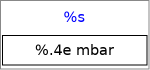
VISUALIZATION TEMPLATE_AMBIENT_PRESSURE_READING  // 150x70
VAR_IN_OUT
	m_instance: FB_METIS_AMBIENT_PRESSURE_SENSOR;
END_VAR
    Rectangle (2,35 145x30), "%.4e mbar", tooltip "Pressure in mbar", text variable: m_instance.stat.lrPressure, colour toggle: NOT m_instance.stat.bValid
    Rectangle (2,2 145x30), "%s", text variable: m_instance.in_sName
END_VISUALIZATION

// HMI/VISUs/Templates/TEMPLATE_BACKGROUND_LEVEL_2
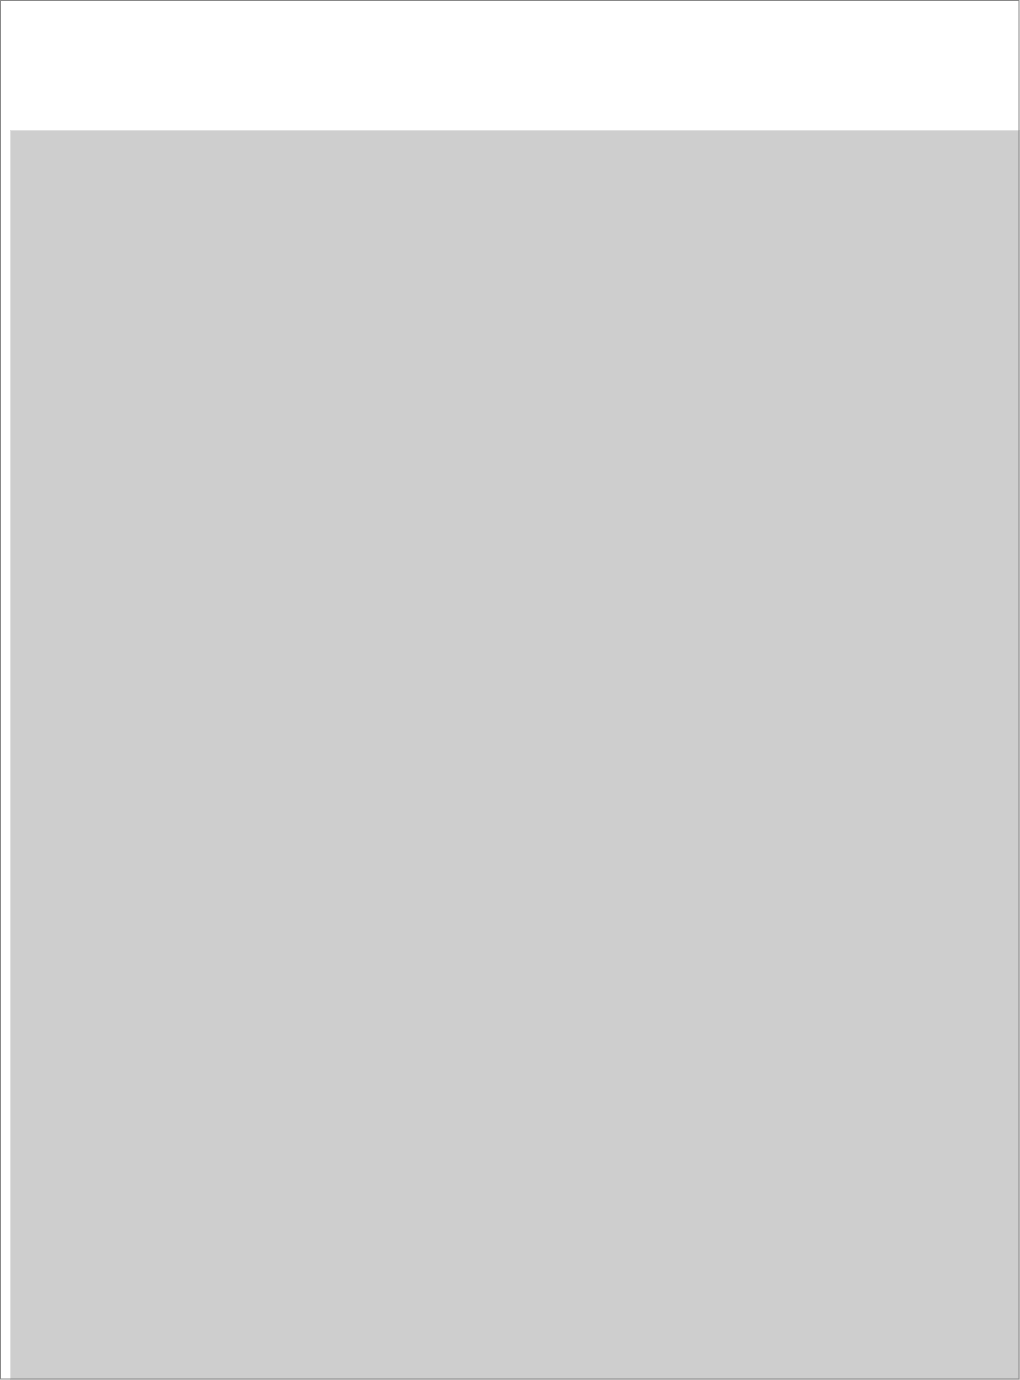
VISUALIZATION TEMPLATE_BACKGROUND_LEVEL_2  // 1020x1380
    Rectangle (10,130 1010x1250)
END_VISUALIZATION

// HMI/VISUs/Templates/TEMPLATE_BACKGROUND_LEVEL_3
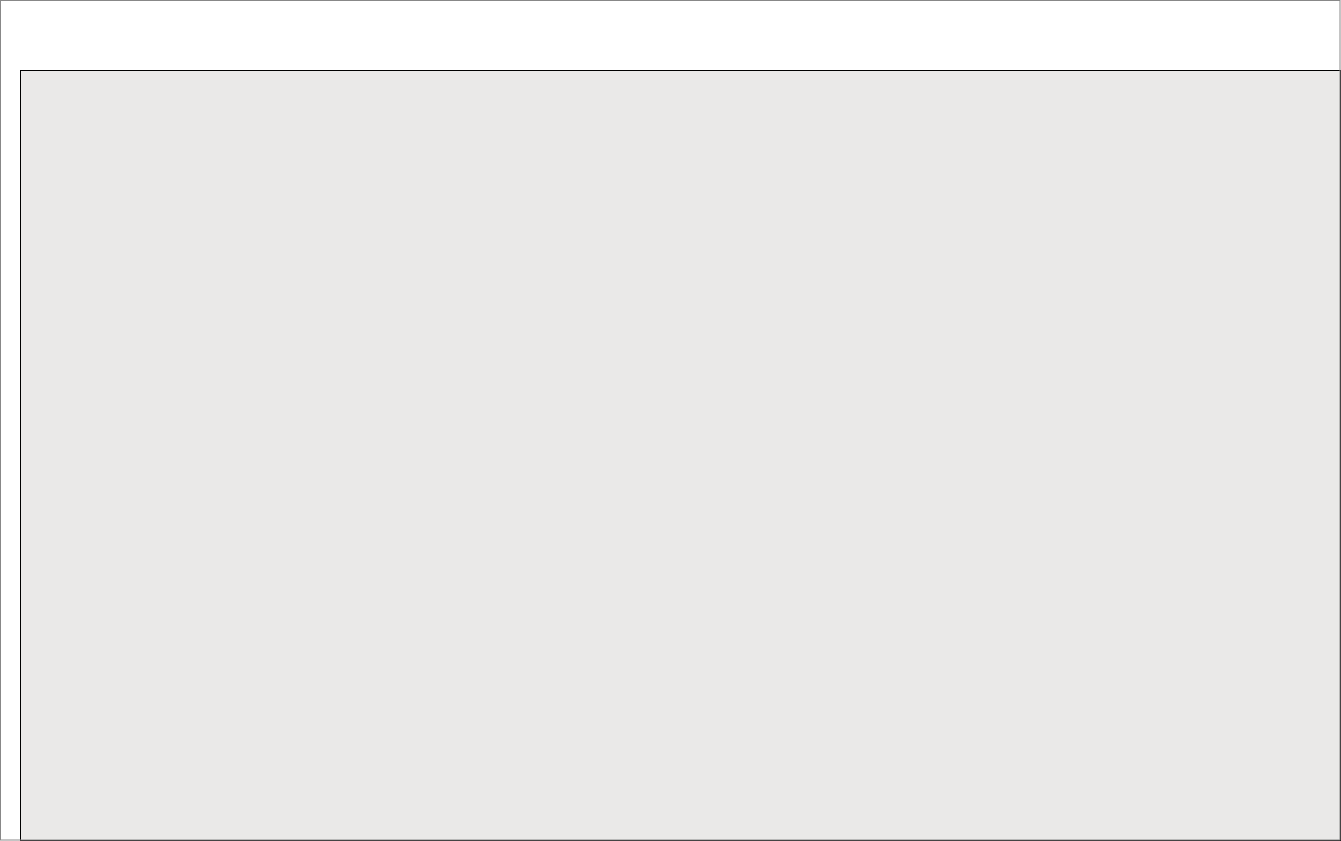
VISUALIZATION TEMPLATE_BACKGROUND_LEVEL_3  // 1341x841
    Rectangle (20,70 1321x771)
END_VISUALIZATION

// HMI/VISUs/Templates/TEMPLATE_BINARY_VALVES
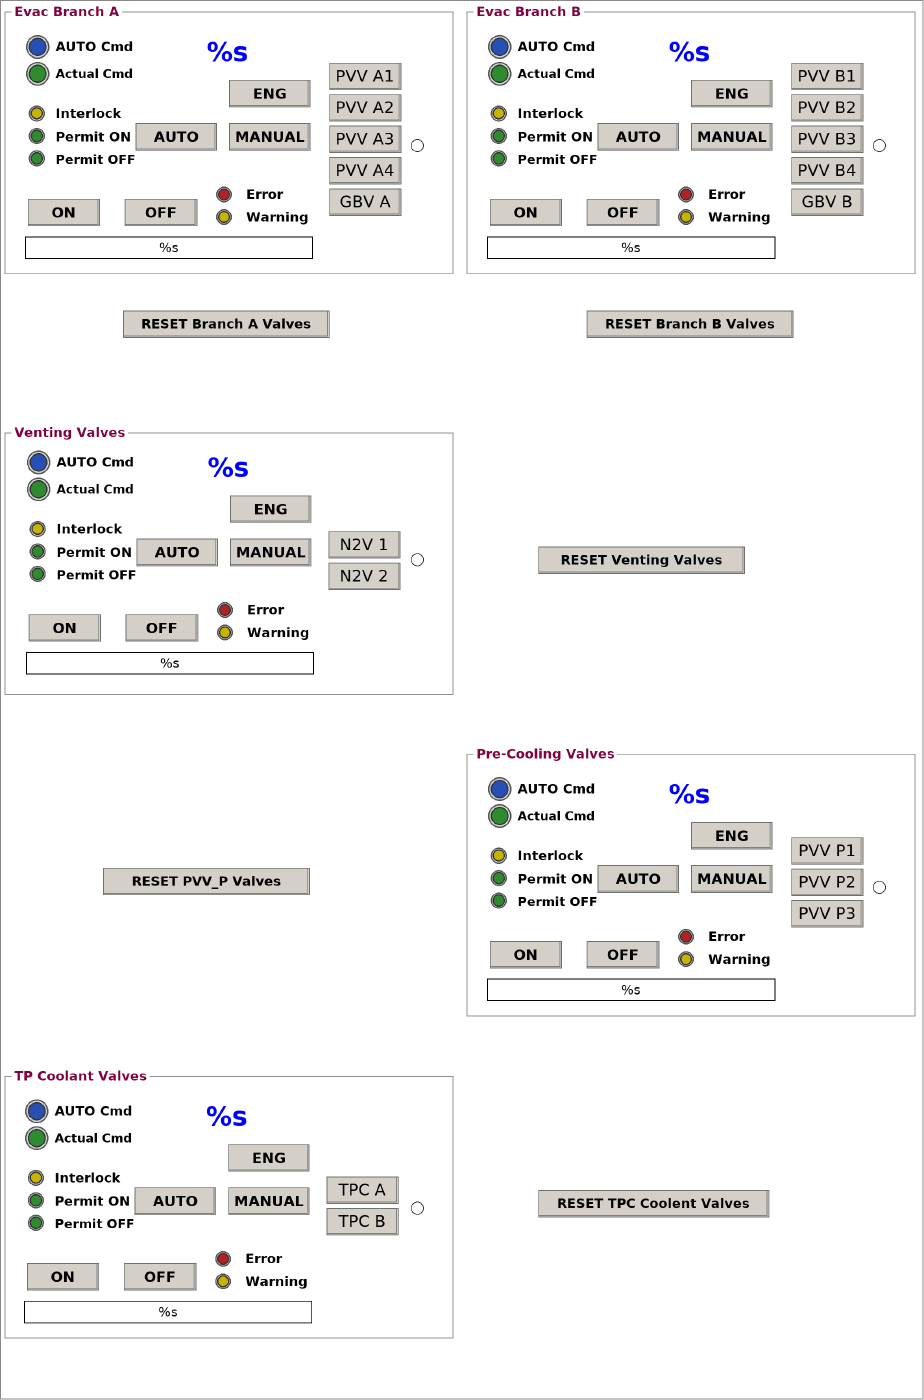
VISUALIZATION TEMPLATE_BINARY_VALVES  // 1030x1560
VAR_IN_OUT
	m_evac_Instance: FB_METIS_CRYO_EVAC;
	m_venting_instance:	FB_METIS_CRYO_VENTING;
	m_cool_down_instance: FB_METIS_CRYO_COOL_DOWN;
	m_cryo_instance:	FB_METIS_CRYO_CTRL;
	
END_VAR
    GroupBox (5,5 500x300), "Evac Branch A"
        Group (18,28 465x255)
            Group (344,37 121x181)
                Button (0,0 80x30), "PVV A1"
                    OnMouseClick: execute { m_evac_Instance.evac_branch_a.guiValveIndex := 1; }
                Button (0,35 80x30), "PVV A2"
                    OnMouseClick: execute { m_evac_Instance.evac_branch_a.guiValveIndex := 2; }
                Button (0,70 80x30), "PVV A3"
                    OnMouseClick: execute { m_evac_Instance.evac_branch_a.guiValveIndex := 3; }
                Button (0,105 80x30), "PVV A4"
                    OnMouseClick: execute { m_evac_Instance.evac_branch_a.guiValveIndex := 4; }
                Button (0,140 80x30), "GBV A"
                    OnMouseClick: execute { m_evac_Instance.evac_branch_a.guiValveIndex := 5; }
                RadioButton (89,3 32x178), variable: m_evac_Instance.evac_branch_a.guiValveIndex-1
            Frame (0,0 326x255)
                shows TEMPLATE_METIS_CMD_OVERRIDE(m_Cmd := m_evac_Instance.evac_branch_a.ptrVC[m_evac_Instance.evac_branch_a.guiValveIndex]^)
    GroupBox (520,5 500x300), "Evac Branch B"
        Group (18,28 465x255)
            Frame (0,0 326x255)
                shows TEMPLATE_METIS_CMD_OVERRIDE(m_Cmd := m_evac_Instance.evac_branch_b.ptrVC[m_evac_Instance.evac_branch_b.guiValveIndex]^)
            Group (344,37 121x181)
                Button (0,0 80x30), "PVV B1"
                    OnMouseClick: execute { m_evac_Instance.evac_branch_b.guiValveIndex := 1; }
                Button (0,35 80x30), "PVV B2"
                    OnMouseClick: execute { m_evac_Instance.evac_branch_b.guiValveIndex := 2; }
                Button (0,70 80x30), "PVV B3"
                    OnMouseClick: execute { m_evac_Instance.evac_branch_b.guiValveIndex := 3; }
                Button (0,105 80x30), "PVV B4"
                    OnMouseClick: execute { m_evac_Instance.evac_branch_b.guiValveIndex := 4; }
                Button (0,140 80x30), "GBV B"
                    OnMouseClick: execute { m_evac_Instance.evac_branch_b.guiValveIndex := 5; }
                RadioButton (89,3 32x178), variable: m_evac_Instance.evac_branch_b.guiValveIndex-1
    GroupBox (520,832 500x300), "Pre-Cooling Valves"
        Group (18,28 465x255)
            Frame (0,0 326x255)
                shows TEMPLATE_METIS_CMD_OVERRIDE(m_Cmd := m_cool_down_instance.ptrVC[m_cool_down_instance.guiValveIndex]^)
            Group (344,73 121x108)
                Button (0,0 80x30), "PVV P1"
                    OnMouseClick: execute { m_cool_down_instance.guiValveIndex := 1; }
                Button (0,35 80x30), "PVV P2"
                    OnMouseClick: execute { m_cool_down_instance.guiValveIndex := 2; }
                RadioButton (89,3 32x105), variable: m_cool_down_instance.guiValveIndex-1
                Button (0,70 80x30), "PVV P3"
                    OnMouseClick: execute { m_cool_down_instance.guiValveIndex := 3; }
    GroupBox (5,474 500x300), "Venting Valves"
        Group (19,22 462x255)
            Frame (0,0 326x255)
                shows TEMPLATE_METIS_CMD_OVERRIDE(m_Cmd := m_venting_instance.ptrVC[m_venting_instance.guiValveIndex]^)
            Group (342,94 120x67)
                Button (0,2 80x30), "N2V 1"
                    OnMouseClick: execute { m_venting_instance.guiValveIndex := 1; }
                Button (0,37 80x30), "N2V 2"
                    OnMouseClick: execute { m_venting_instance.guiValveIndex := 2; }
                RadioButton (90,0 30x67), variable: m_venting_instance.guiValveIndex-1
                    Areas[0]: Text=Radiobutton
                    Areas[1]: Text=Radiobutton
    GroupBox (5,1191 500x300), "TP Coolant Valves"
        Frame (17,28 326x255)
            shows TEMPLATE_METIS_CMD_OVERRIDE(m_Cmd := m_cryo_instance.ptrVC[m_cryo_instance.guiCoolantValveIndex]^)
        Group (359,120 124x70)
            Button (0,0 80x30), "TPC A"
                OnMouseClick: execute { m_cryo_instance.guiCoolantValveIndex := 1; }
            Button (0,35 80x30), "TPC B"
                OnMouseClick: execute { m_cryo_instance.guiCoolantValveIndex := 2; }
            RadioButton (92,0 32x70), variable: m_cryo_instance.guiCoolantValveIndex-1
    Button (137,346 230x30), "RESET Branch A Valves"
        OnMouseClick: execute { m_evac_Instance.evac_branch_a.bReset_Valves := TRUE; }
    Button (654,346 230x30), "RESET Branch B Valves"
        OnMouseClick: execute { m_evac_Instance.evac_branch_b.bReset_Valves := TRUE; }
    Button (600,609 230x30), "RESET Venting Valves"
        OnMouseClick: execute { m_venting_instance.bReset_Valves := TRUE; }
    Button (115,967 230x30), "RESET PVV_P Valves"
        OnMouseClick: execute { m_cool_down_instance.bReset_Valves := TRUE; }
    Button (600,1326 257x30), "RESET TPC Coolent Valves"
        OnMouseClick: execute { m_cryo_instance.TPC_A.M_Reset(); m_cryo_instance.TPC_B.M_Reset(); }
END_VISUALIZATION

// HMI/VISUs/Templates/TEMPLATE_CRYO_SENSOR_TEMPERATURE
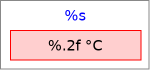
VISUALIZATION TEMPLATE_CRYO_SENSOR_TEMPERATURE  // 150x70
VAR_IN_OUT
	m_instance:	FB_CRYO_SENSOR_TEMPERATURE;
END_VAR
    Rectangle (10,30 131x30)
    Rectangle (10,30 131x30), invisible if: NOT m_instance.stat.bError
    Rectangle (10,30 131x31), "%.2f °C", text variable: m_instance.stat.lrTempC
    Rectangle (0,0 151x31), "%s", text variable: m_instance.in_sName
END_VISUALIZATION

// HMI/VISUs/Templates/TEMPLATE_EVACUATION
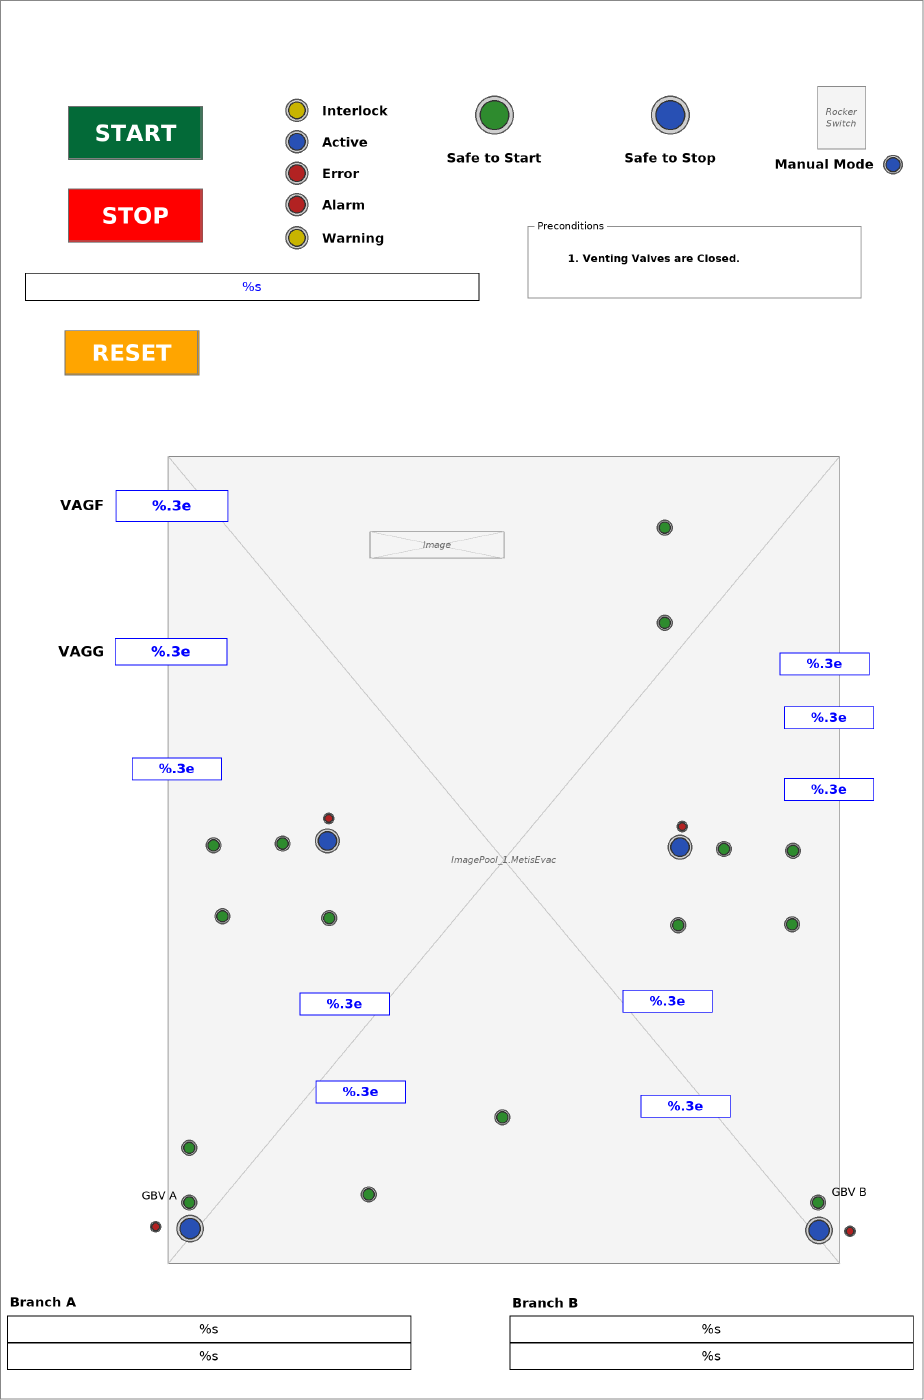
VISUALIZATION TEMPLATE_EVACUATION  // 1030x1560
VAR_IN_OUT
	m_Instance: FB_METIS_CRYO_EVAC;
	m_venting_instance:	FB_METIS_CRYO_VENTING;
	m_cool_down_instance: FB_METIS_CRYO_COOL_DOWN;
	
END_VAR
    Group (8,508 1010x1018)
        Group (0,928 1010x90)
            Group (0,0 450x90)
                Rectangle (0,30 450x30), "%s", text variable: m_Instance.evac_branch_a.stat.sErrorText
                Rectangle (0,60 450x30), "%s", text variable: m_Instance.evac_branch_a.stat.sStatus
                Rectangle (0,0 100x30), "Branch A"
            Group (560,1 450x89)
                Rectangle (0,29 450x30), "%s", text variable: m_Instance.evac_branch_b.stat.sErrorText
                Rectangle (0,59 450x30), "%s", text variable: m_Instance.evac_branch_b.stat.sStatus
                Rectangle (0,0 100x30), "Branch B"
        Group (45,0 921x900)
            Image (134,0 749x900), image: ImagePool_1.MetisEvac
            Image (359,84 150x30)
            Rectangle (281,598 100x25), "%.3e", text variable: m_Instance.evac_branch_a.VAG1.stat.lrPressure
            Rectangle (94,336 100x25), "%.3e", text variable: m_Instance.evac_branch_a.VAG2.stat.lrPressure
            Lamp1 (141,843 36x36), variable: m_Instance.evac_branch_a.rp.stat.bReady, style: Lamp-Lamp1-Blue
            Lamp1 (296,413 32x32), tooltip "If ON, TMP pump is at its nominal speed, i.e. Ready.", variable: m_Instance.evac_branch_a.tp.stat.bReady, style: Lamp-Lamp1-Blue
            Lamp1 (185,503 20x20), variable: m_Instance.evac_branch_a.PVV1.stat.bActON, style: Lamp-Lamp1-Green
            Lamp1 (304,505 20x20), variable: m_Instance.evac_branch_a.PVV2.stat.bActON, style: Lamp-Lamp1-Green
            Lamp1 (175,424 20x20), variable: m_Instance.evac_branch_a.PVV3.stat.bActON, style: Lamp-Lamp1-Green
            Lamp1 (252,422 20x20), variable: m_Instance.evac_branch_a.PVV4.stat.bActON, style: Lamp-Lamp1-Green
            Lamp1 (148,822 20x20), variable: m_Instance.evac_branch_a.GBV.stat.bActON, style: Lamp-Lamp1-Green
            Lamp1 (306,397 15x14), tooltip "If ON, TMP pump is still spinning.", variable: m_Instance.evac_branch_a.tp.stat.bSpeed100, style: Lamp-Lamp1-Red
            Rectangle (299,696 100x25), "%.3e", text variable: m_Instance.evac_branch_a.VAG3.stat.lrPressure
            Lamp1 (689,420 32x32), tooltip "If ON, TMP pump is at its nominal speed, i.e. Ready.", variable: m_Instance.evac_branch_b.tp.stat.bReady, style: Lamp-Lamp1-Blue
            Lamp1 (700,406 15x14), tooltip "If ON, TMP pump is still spinning.", variable: m_Instance.evac_branch_b.tp.stat.bSpeed100, style: Lamp-Lamp1-Red
            Lamp1 (744,428 20x20), variable: m_Instance.evac_branch_b.PVV4.stat.bActON, style: Lamp-Lamp1-Green
            Lamp1 (821,430 20x20), variable: m_Instance.evac_branch_b.PVV3.stat.bActON, style: Lamp-Lamp1-Green
            Lamp1 (693,513 20x20), variable: m_Instance.evac_branch_b.PVV2.stat.bActON, style: Lamp-Lamp1-Green
            Lamp1 (820,512 20x20), variable: m_Instance.evac_branch_b.PVV1.stat.bActON, style: Lamp-Lamp1-Green
            Lamp1 (842,845 36x36), variable: m_Instance.evac_branch_b.rp.stat.bReady, style: Lamp-Lamp1-Blue
            Lamp1 (849,822 20x20), variable: m_Instance.evac_branch_b.GBV.stat.bActON, style: Lamp-Lamp1-Green
            Rectangle (661,712 100x25), "%.3e", text variable: m_Instance.evac_branch_b.VAG3.stat.lrPressure
            Rectangle (821,359 100x25), "%.3e", text variable: m_Instance.evac_branch_b.VAG2.stat.lrPressure
            Rectangle (641,595 100x25), "%.3e", text variable: m_Instance.evac_branch_b.VAG1.stat.lrPressure
            Lamp1 (678,70 20x20), variable: m_venting_instance.N2V_1.stat.bActON, style: Lamp-Lamp1-Green
            Lamp1 (678,176 20x20), variable: m_venting_instance.N2V_2.stat.bActON, style: Lamp-Lamp1-Green
            Lamp1 (148,761 20x20), variable: m_cool_down_instance.PVV_P1.stat.bActON, style: Lamp-Lamp1-Green
            Lamp1 (348,813 20x20), variable: m_cool_down_instance.PVV_P3.stat.bActON, style: Lamp-Lamp1-Green
            Lamp1 (497,727 20x20), variable: m_cool_down_instance.PVV_P2.stat.bActON, style: Lamp-Lamp1-Green
            Rectangle (97,809 55x30), "GBV A"
            Rectangle (866,805 55x30), "GBV B"
            Group (1,38 200x35)
                Rectangle (75,0 125x35), "%.3e", text variable: m_Instance.VAGF.stat.lrPressure
                Rectangle (0,2 75x30), "VAGF"
            Group (0,203 200x30)
                Rectangle (75,0 125x30), "%.3e", text variable: m_Instance.VAGG.stat.lrPressure
                Rectangle (0,0 75x30), "VAGG"
            Rectangle (816,219 100x25), "%.3e", text variable: m_venting_instance.sensor_HPG1.stat.lrPressure
            Rectangle (821,279 100x25), "%.3e", text variable: m_venting_instance.sensor_HPG2.stat.lrPressure
    Group (76,118 150x152)
        Button (0,0 150x60), "START", input disabled if: NOT m_Instance.in_Cryo_Stat.bVentingValvesAreClosed
            OnMouseClick: execute { m_Instance.ctrl.bEnable := TRUE; }
        Button (0,92 150x60), "STOP", input disabled if: (NOT m_instance.in_Cryo_Stat.bPermitEvacuationStop) AND (NOT m_Instance.stat.bManual)
            OnMouseClick: execute { m_Instance.ctrl.bEnable := FALSE; }
    Group (316,108 131x173)
        Group (0,35 131x31)
            Label (40,0 91x31), "Active"
            Lamp1 (0,0 30x30), variable: m_Instance.stat.bActive, style: Lamp-Lamp1-Blue
        Group (0,70 130x31)
            Label (40,0 90x31), "Error"
            Lamp1 (0,0 30x30), variable: m_Instance.stat.bError, style: Lamp-Lamp1-Red
        Group (0,0 131x31)
            Lamp1 (0,0 30x30), variable: m_Instance.interlocks.bInterlock_Evacuation, style: Lamp-Lamp1-Yellow
            Label (40,0 91x31), "Interlock"
        Group (0,105 130x31)
            Label (40,0 90x31), "Alarm"
            Lamp1 (0,0 30x30), variable: m_Instance.stat.bAlarm, style: Lamp-Lamp1-Red
        Group (0,142 130x31)
            Label (40,0 90x31), "Warning"
            Lamp1 (0,0 30x30), variable: m_Instance.stat.bWarning, style: Lamp-Lamp1-Yellow
    Group (672,103 150x88)
        Lamp1 (50,0 50x50), variable: m_Instance.in_Cryo_Stat.bPermitEvacuationStop, style: Lamp-Lamp1-Blue
        Rectangle (0,58 150x30), "Safe to Stop"
    GroupBox (588,244 372x88), "Preconditions"
        Rectangle (42,29 300x30), "1. Venting Valves are Closed.", colour toggle: m_Instance.in_Cryo_Stat.bVentingValvesAreClosed
    Button (72,368 150x50), "RESET", invisible if: NOT m_Instance.stat.bError
        OnMouseClick: execute { m_Instance.ctrl.bReset := TRUE; }
    Rectangle (28,304 506x31), "%s", text variable: m_instance.stat.sState
    Group (868,168 140x30)
        Label (0,0 109x30), "Manual Mode"
        Lamp1 (115,3 25x25), variable: m_Instance.stat.bManual, style: Lamp-Lamp1-Blue
    RockerSwitch (911,96 54x70), tooltip "Activates the Manual mode", variable: m_Instance.stat.bManual, input disabled if: m_Instance.stat.bVentingValvesOpen, behaviour: TOGGLE, style: Switch-RockerSwitch-Red
    Group (476,103 150x88)
        Lamp1 (50,0 50x50), variable: NOT m_Instance.interlocks.bInterlock_Evacuation, style: Lamp-Lamp1-Green
        Rectangle (0,58 150x30), "Safe to Start"
    Lamp1 (940,1365 15x14), tooltip "If ON, RP pump is still spinning.", variable: m_Instance.evac_branch_b.rp.stat.bMoving, style: Lamp-Lamp1-Red
    Lamp1 (166,1360 15x14), tooltip "If ON, RP pump is still spinning.", variable: m_Instance.evac_branch_a.rp.stat.bMoving, style: Lamp-Lamp1-Red
END_VISUALIZATION

// HMI/VISUs/Templates/TEMPLATE_HEATER_CPAU60
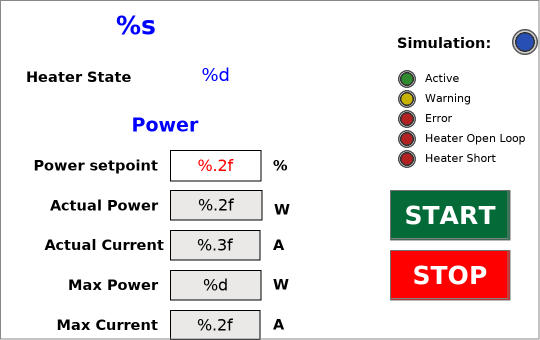
VISUALIZATION TEMPLATE_HEATER_CPAU60  // 540x340
VAR_IN_OUT
	m_instance: FB_HEATER_CPAU60;
	m_bEnable:	BOOL;	// Flag to start/stop the Heater
END_VAR
    Rectangle (21,10 230x30), "%s", text variable: m_Instance.in_sName
    Button (390,190 120x50), "START"
        OnMouseClick: execute { m_bEnable := TRUE; }
    Button (390,250 120x50), "STOP"
        OnMouseClick: execute { m_bEnable := FALSE; }
    Lamp1 (397,69 20x20), tooltip "If ON, Heater is active", variable: m_Instance.stat.bActive, style: Lamp-Lamp1-Green
    Lamp1 (397,89 20x20), tooltip "If ON, reading is in Warning", variable: m_Instance.stat.bWarning, style: Lamp-Lamp1-Yellow
    Lamp1 (397,129 20x20), tooltip "If ON, Heater circuit is open", variable: m_Instance.stat.bHeaterOpenLoop, style: Lamp-Lamp1-Red
    Lamp1 (397,149 20x20), tooltip "If ON, Heater is in short circuit", variable: m_Instance.stat.bHeaterShort, style: Lamp-Lamp1-Red
    Lamp1 (397,109 20x20), tooltip "If ON, reading is in error.", variable: m_Instance.stat.bError, style: Lamp-Lamp1-Red
    Label (422,67 87x23), "Active"
    Label (422,87 87x23), "Warning"
    Label (422,107 87x23), "Error"
    Label (422,127 112x23), "Heater Open Loop"
    Label (422,147 87x23), "Heater Short"
    Rectangle (170,150 91x31), "%.2f", tooltip "Simulated value [K] when simulation is active.", text variable: m_instance.ctrl.lrPower, input disabled if: Not m_instance.bManualInputFlag
        OnMouseClick: write the text variable via Default
    Rectangle (170,190 92x30), "%.2f", tooltip "Value used by the system [K]", text variable: m_instance.stat.lrActHeaterPower
    Rectangle (170,230 90x30), "%.3f", tooltip "Value used by the system [C]", text variable: m_instance.stat.lrActCurrent
    Lamp1 (510,27 30x30), tooltip "If ON, Heater is simulated.", variable: m_instance.stat.bSimulated, style: Lamp-Lamp1-Blue
    Rectangle (394,28 110x30), "Simulation:"
    Rectangle (90,110 150x30), "Power"
    Rectangle (271,195 29x29), "W"
    Rectangle (270,230 32x30), "A"
    Rectangle (138,60 156x30), "%d", text variable: m_Instance.stat.nHeaterState
    Rectangle (23,62 110x30), "Heater State"
    Rectangle (30,150 131x31), "Power setpoint"
    Rectangle (50,190 111x31), "Actual Power"
    Rectangle (270,150 29x31), "%"
    Rectangle (40,230 127x30), "Actual Current"
    Rectangle (170,270 91x30), "%d", tooltip "Value used by the system [K]", text variable: m_instance.in_nMaxHeaterPower
    Rectangle (170,310 90x30), "%.2f", tooltip "Value used by the system [K]", text variable: m_instance.stat.lrMaxCurrent
    Rectangle (60,270 101x30), "Max Power"
    Rectangle (30,310 131x30), "Max Current"
    Rectangle (270,270 29x29), "W"
    Rectangle (270,310 29x29), "A"
END_VISUALIZATION

// HMI/VISUs/Templates/TEMPLATE_HEATER_CXWUI60
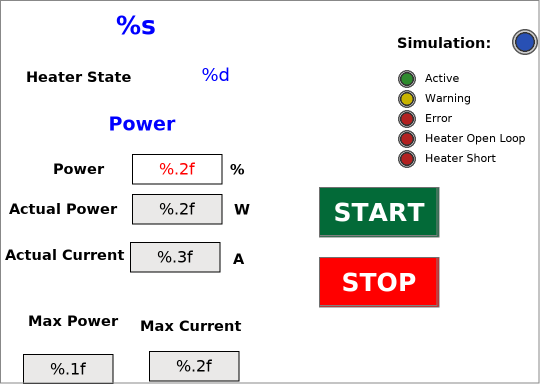
VISUALIZATION TEMPLATE_HEATER_CXWUI60  // 540x384
VAR_IN_OUT
	m_instance: FB_HEATER_CXWUI60;
	m_bEnable:	BOOL;	// Flag to start/stop the Heater
END_VAR
    Rectangle (21,10 230x30), "%s", text variable: m_Instance.in_sName
    Button (319,187 120x50), "START"
        OnMouseClick: execute { m_bEnable := TRUE; }
    Button (319,257 120x50), "STOP"
        OnMouseClick: execute { m_bEnable := FALSE; }
    Lamp1 (397,69 20x20), tooltip "If ON, Heater is active", variable: m_Instance.stat.bActive, style: Lamp-Lamp1-Green
    Lamp1 (397,89 20x20), tooltip "If ON, reading is in Warning", variable: m_Instance.stat.bWarning, style: Lamp-Lamp1-Yellow
    Lamp1 (397,129 20x20), tooltip "If ON, Heater circuit is open", variable: m_Instance.stat.bHeaterOpenLoop, style: Lamp-Lamp1-Red
    Lamp1 (397,149 20x20), tooltip "If ON, Heater is in short circuit", variable: m_Instance.stat.bHeaterShort, style: Lamp-Lamp1-Red
    Lamp1 (397,109 20x20), tooltip "If ON, reading is in error.", variable: m_Instance.stat.bError, style: Lamp-Lamp1-Red
    Label (422,67 87x23), "Active"
    Label (422,87 87x23), "Warning"
    Label (422,107 87x23), "Error"
    Label (422,127 112x23), "Heater Open Loop"
    Label (422,147 87x23), "Heater Short"
    Rectangle (132,154 90x30), "%.2f", tooltip "Simulated value [K] when simulation is active.", text variable: m_instance.ctrl.lrPower, input disabled if: Not m_instance.bManualInputFlag
        OnMouseClick: write the text variable via Default
    Rectangle (132,194 90x30), "%.2f", tooltip "Value used by the system [K]", text variable: m_instance.stat.lrActHeaterPower
    Rectangle (130,242 90x30), "%.3f", tooltip "Value used by the system [C]", text variable: m_instance.stat.lrActCurrent
    Lamp1 (510,27 30x30), tooltip "If ON, Heater is simulated.", style: Lamp-Lamp1-Blue
    Rectangle (394,28 110x30), "Simulation:"
    Rectangle (67,109 150x30), "Power"
    Rectangle (231,195 29x29), "W"
    Rectangle (230,244 32x30), "A"
    Rectangle (138,60 156x30), "%d", text variable: m_Instance.stat.nHeaterState
    Rectangle (23,62 110x30), "Heater State"
    Rectangle (50,154 66x30), "Power"
    Rectangle (6,194 110x30), "Actual Power"
    Rectangle (227,155 29x29), "%"
    Rectangle (2,240 127x30), "Actual Current"
    Rectangle (23,354 90x30), "%.1f", tooltip "Value used by the system [K]", text variable: m_instance.in_nMaxHeaterPower
    Rectangle (149,351 90x30), "%.2f", tooltip "Value used by the system [K]", text variable: m_instance.stat.lrMaxCurrent
    Rectangle (25,306 92x30), "Max Power"
    Rectangle (137,311 127x30), "Max Current"
END_VISUALIZATION

// HMI/VISUs/Templates/TEMPLATE_HEATER_PWM_CTRL
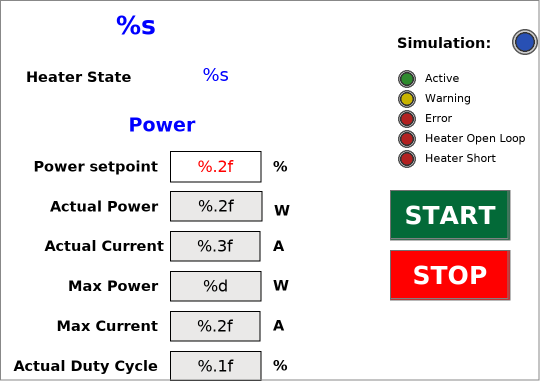
VISUALIZATION TEMPLATE_HEATER_PWM_CTRL  // 540x381
VAR_IN_OUT
	m_instance: FB_HEATER_PWM;
	m_bEnable:	BOOL;	// Flag to start/stop the Heater
END_VAR
    Rectangle (170,351 91x30), "%.1f", tooltip "Value used by the system [C]", text variable: m_instance.stat.lrActDutyCycle
    Rectangle (10,351 151x30), "Actual Duty Cycle"
    Rectangle (21,10 230x30), "%s", text variable: m_Instance.in_sName
    Button (390,190 120x50), "START"
        OnMouseClick: execute { m_bEnable := TRUE; }
    Button (390,250 120x50), "STOP"
        OnMouseClick: execute { m_bEnable := FALSE; }
    Lamp1 (397,69 20x20), tooltip "If ON, Heater is active", variable: m_Instance.stat.bActive, style: Lamp-Lamp1-Green
    Lamp1 (397,89 20x20), tooltip "If ON, reading is in Warning", variable: m_Instance.stat.bWarning, style: Lamp-Lamp1-Yellow
    Lamp1 (397,129 20x20), tooltip "If ON, Heater circuit is open", variable: m_Instance.stat.bHeaterOpenLoop, style: Lamp-Lamp1-Red
    Lamp1 (397,149 20x20), tooltip "If ON, Heater is in short circuit", variable: m_Instance.stat.bHeaterShort, style: Lamp-Lamp1-Red
    Lamp1 (397,109 20x20), tooltip "If ON, reading is in error.", variable: m_Instance.stat.bError, style: Lamp-Lamp1-Red
    Label (422,67 87x23), "Active"
    Label (422,87 87x23), "Warning"
    Label (422,107 87x23), "Error"
    Label (422,127 112x23), "Heater Open Loop"
    Label (422,147 87x23), "Heater Short"
    Rectangle (170,151 91x31), "%.2f", tooltip "Simulated value [K] when simulation is active.", text variable: m_instance.ctrl.lrPower, input disabled if: Not m_instance.bManualInputFlag
        OnMouseClick: write the text variable via Default
    Rectangle (170,191 92x30), "%.2f", tooltip "Value used by the system [K]", text variable: m_instance.stat.lrActHeaterPower
    Rectangle (170,231 90x30), "%.3f", tooltip "Value used by the system [C]", text variable: m_instance.stat.lrActCurrent
    Lamp1 (510,27 30x30), tooltip "If ON, Heater is simulated.", variable: m_instance.stat.bSimulated, style: Lamp-Lamp1-Blue
    Rectangle (394,28 110x30), "Simulation:"
    Rectangle (87,110 150x30), "Power"
    Rectangle (271,196 29x29), "W"
    Rectangle (270,231 32x30), "A"
    Rectangle (138,60 156x30), "%s", text variable: m_Instance.stat.sHeaterState
    Rectangle (23,62 110x30), "Heater State"
    Rectangle (30,151 131x31), "Power setpoint"
    Rectangle (50,191 111x31), "Actual Power"
    Rectangle (270,151 29x31), "%"
    Rectangle (40,231 127x30), "Actual Current"
    Rectangle (170,271 91x30), "%d", tooltip "Value used by the system [K]", text variable: m_instance.in_nMaxHeaterPower
    Rectangle (170,311 90x30), "%.2f", tooltip "Value used by the system [K]", text variable: m_instance.stat.lrMaxCurrent
    Rectangle (60,271 101x30), "Max Power"
    Rectangle (30,311 131x30), "Max Current"
    Rectangle (270,271 29x29), "W"
    Rectangle (270,311 29x29), "A"
    Rectangle (270,350 29x31), "%"
END_VISUALIZATION

// HMI/VISUs/Templates/TEMPLATE_LN2_LEVEL_SENSOR_AND_CTRL
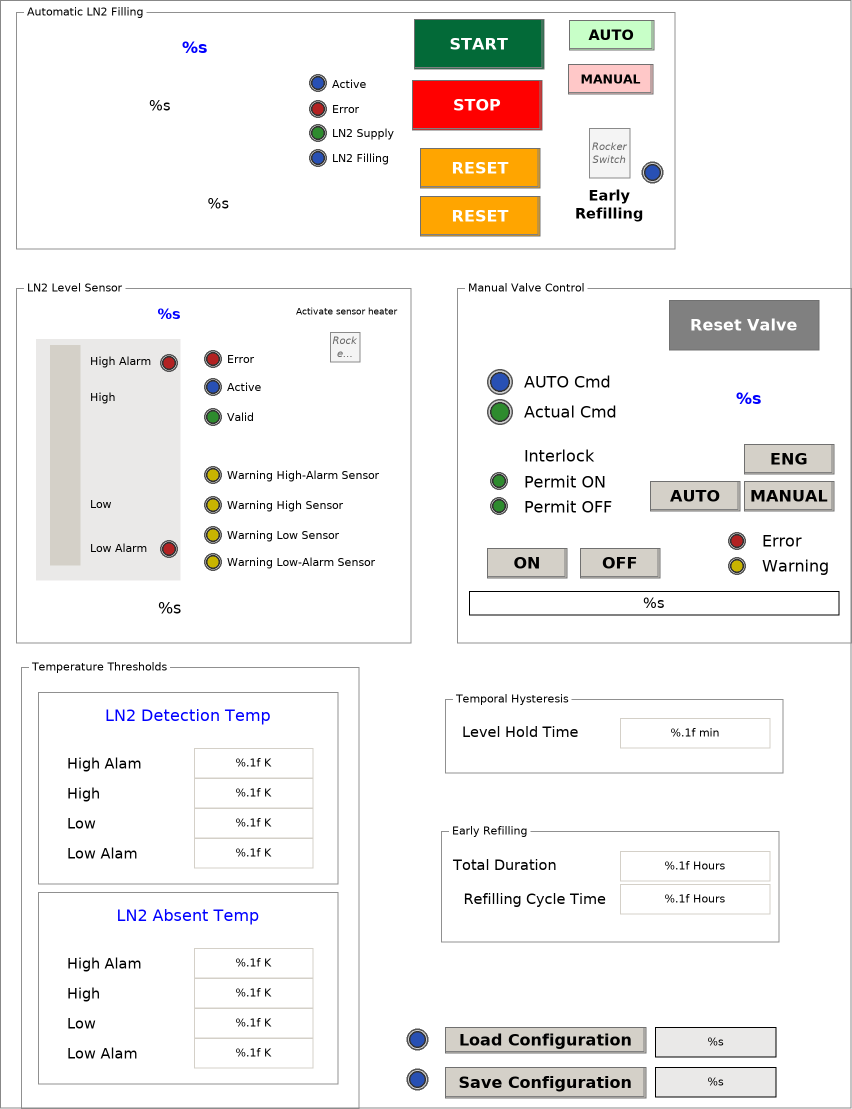
VISUALIZATION TEMPLATE_LN2_LEVEL_SENSOR_AND_CTRL  // 852x1109
VAR_IN_OUT
	m_level_control_instance: FB_METIS_CRYO_LN2_LEVEL_CTRL;
	m_instance: FB_METIS_CRYO_LN2_SENSOR;
	m_cmd: FB_CRYO_CMD_OVERRIDE;
	m_bEnable:	BOOL;	// Flag to start/stop LN2 level control
END_VAR
    GroupBox (457,280 395x363), "Manual Valve Control"
        Button (212,20 150x50), "Reset Valve", tooltip "Reset LN2 filling valve"
            OnMouseClick: execute { m_level_control_instance.M_ResetValve(); }
    Group (469,367 370x248)
        Lamp1 (20,104 20x20), variable: m_Cmd.bPermitOn, style: Lamp-Lamp1-Green
        Lamp1 (20,129 20x20), variable: m_Cmd.bPermitOff, style: Lamp-Lamp1-Green
        Rectangle (52,74 110x30), "Interlock"
        Rectangle (52,100 110x30), "Permit ON"
        Rectangle (52,125 110x30), "Permit OFF"
        Button (18,181 80x30), "ON", colour toggle: (m_Cmd.bPermitOn AND NOT m_Cmd.bAutoMode) OR m_Cmd.bEngMode, input disabled if: m_Cmd.bDisableBtnOn
            OnMouseClick: execute { m_Cmd.bManualCmd := TRUE; }
        Lamp1 (16,30 30x30), tooltip "Actual command going out", variable: m_Cmd.out_bEnable, style: Lamp-Lamp1-Green
        Rectangle (52,30 110x30), "Actual Cmd"
        Button (181,114 90x30), "AUTO", tooltip "Switch to AUTO Mode", colour toggle: m_Cmd.bAutoMode, input disabled if: m_Cmd.bAutoMode OR m_Cmd.bEngMode
            OnMouseClick: execute { m_Cmd.bAutoMode := TRUE; }
        Button (275,114 90x30), "MANUAL", tooltip "Switch to MANUAL Mode", colour toggle: NOT m_Cmd.bAutoMode, input disabled if: NOT m_Cmd.bAutoMode AND NOT m_Cmd.bEngMode
            OnMouseClick: execute { m_Cmd.bAutoMode := FALSE; }
        Button (111,181 80x30), "OFF", colour toggle: (m_Cmd.bPermitOff AND NOT m_Cmd.bAutoMode) OR m_Cmd.bEngMode, input disabled if: m_Cmd.bDisableBtnOff
            OnMouseClick: execute { m_Cmd.bManualCmd := FALSE; }
        Button (275,77 90x30), "ENG", tooltip "Toggle Engineering Mode", colour toggle: m_Cmd.bEngMode, input disabled if: m_Cmd.bAutoMode
            toggle m_Cmd.bEngMode
        Lamp1 (16,0 30x30), tooltip "Command coming from the Control System", variable: m_Cmd.in_bEnable, style: Lamp-Lamp1-Blue
        Rectangle (52,0 110x30), "AUTO Cmd"
        Rectangle (0,224 370x24), "%s", text variable: m_Cmd.out_sStatus
        Lamp1 (258,164 20x20), tooltip "If ON, there is an error in the SW implementation of permission handling.", variable: m_Cmd.out_bError, style: Lamp-Lamp1-Red
        Rectangle (290,159 75x30), "Error"
        Lamp1 (258,189 20x20), tooltip "If ON, ENG command is not safe!", variable: m_Cmd.out_bWarning, style: Lamp-Lamp1-Yellow
        Rectangle (290,184 75x30), "Warning"
        Rectangle (205,11 150x41), "%s", text variable: m_Cmd.out_sMode
    GroupBox (441,823 338x119), "Early Refilling", tooltip "Time to hold a change of status to avoid transient oscillations."
        Label (9,59 170x34), "Refilling Cycle Time"
        Textfield (179,61 150x30), "%.1f Hours", tooltip "(Hours) Refilling cycle time during the Early refilling", text variable: m_level_control_instance.cfg.lr_Cycle_Time, input disabled if: m_level_control_instance.bAuto
            OnMouseClick: write the text variable via Default
        Textfield (179,28 150x30), "%.1f Hours", tooltip "(Hours) The total duration of Early Refilling", text variable: m_level_control_instance.cfg.lr_Early_Refill_Duration_Time, input disabled if: m_level_control_instance.bAuto
            OnMouseClick: write the text variable via Default
        Label (9,25 170x34), "Total Duration"
    GroupBox (445,691 338x82), "Temporal Hysteresis", tooltip "Time to hold a change of status to avoid transient oscillations."
        Textfield (175,27 150x30), "%.1f min", tooltip "(Minutes) LN2 level hold time to reduce oscilations at level change", text variable: m_level_control_instance.cfg.lr_LN2Level_Hold_Time, input disabled if: m_level_control_instance.bAuto
            OnMouseClick: write the text variable via Default
        Label (14,24 158x34), "Level Hold Time"
    GroupBox (16,4 659x245), "Automatic LN2 Filling"
        Rectangle (12,74 264x55), "%s", text variable: m_level_control_instance.sState
        Label (313,69 46x23), "Active"
        Lamp1 (292,95 20x20), tooltip "pump speed > 0 rpm", variable: m_level_control_instance.bError, style: Lamp-Lamp1-Red
        Label (313,94 46x23), "Error"
        Lamp1 (292,69 20x20), tooltip "pump speed > 0 rpm", variable: m_level_control_instance.bActive, style: Lamp-Lamp1-Blue
        Lamp1 (292,119 20x20), tooltip "pump speed > 0 rpm", variable: m_level_control_instance.in_ESO_LN2_Supply, style: Lamp-Lamp1-Green
        Button (553,16 85x30), "AUTO", tooltip "Automatic LN2 Level Control", colour toggle: m_level_control_instance.bAuto
            OnMouseClick: execute { m_level_control_instance.bManual := FALSE; m_level_control_instance.bAuto := TRUE; }
        Button (552,60 85x30), "MANUAL", tooltip "Manually start/Stop LN2 Level Control", colour toggle: m_level_control_instance.bManual
            OnMouseClick: execute { m_level_control_instance.bManual := TRUE; m_level_control_instance.bAuto := FALSE; }
        Group (552,124 83x97)
            RockerSwitch (21,0 41x50), tooltip "Activate or deactivate early LN2 refilling", variable: m_level_control_instance.bEarly_Refilling, behaviour: TOGGLE, style: Switch-RockerSwitch-Blue
            Label (0,56 83x41), "Early Refilling"
        Button (404,144 120x40), "RESET"
            OnMouseClick: execute {
                m_level_control_instance.nState := E_LN2_LEVEL_CTRL_STATE.ERROR; // RESET
                m_level_control_instance.bReset := TRUE;
            }
        Button (404,192 120x40), "RESET", invisible if: NOT m_level_control_instance.bError
            OnMouseClick: execute { m_level_control_instance.bReset := TRUE; }
        Rectangle (12,172 381x55), "%s", text variable: m_level_control_instance.sSubState
        Lamp1 (292,144 20x20), tooltip "pump speed > 0 rpm", variable: m_level_control_instance.bFilling, style: Lamp-Lamp1-Blue
        Lamp1 (624,156 25x25), tooltip "pump speed > 0 rpm", variable: m_level_control_instance.bEarly_Refilling, style: Lamp-Lamp1-Blue
    GroupBox (16,280 395x363), "LN2 Level Sensor", tooltip "LN2 Level Sensor"
        RockerSwitch (314,52 30x30), tooltip "Activate or deactivate sensor heaters", variable: m_instance.bActivateSensor, behaviour: TOGGLE, style: Switch-RockerSwitch-Yellow
        Label (277,16 111x31), "Activate sensor heater"
    Rectangle (37,299 264x30), "%s", text variable: m_instance.in_sName
    Rectangle (36,339 144x241)
    Group (50,345 30x220)
        Rectangle (0,180 30x40), colour toggle: m_instance.stat.bLowAlarm
        Rectangle (0,110 30x70), colour toggle: m_instance.stat.bLow
        Rectangle (0,40 30x70), colour toggle: m_instance.stat.bHigh
        Rectangle (0,0 30x40), colour toggle: m_instance.stat.bHighAlarm
    Label (87,350 70x23), "High Alarm"
    Label (87,386 34x23), "High"
    Label (87,493 28x23), "Low"
    Label (87,537 70x23), "Low Alarm"
    Lamp1 (159,353 20x20), variable: m_instance.stat.bLowAlarm AND ( m_instance.stat.bLow) AND ( m_instance.stat.bHigh) AND (m_instance.stat.bHighAlarm), style: Lamp-Lamp1-Red
    Lamp1 (159,539 20x20), variable: m_instance.stat.bLowAlarm AND (NOT m_instance.stat.bLow) AND (NOT m_instance.stat.bHigh) AND (NOT m_instance.stat.bHighAlarm), style: Lamp-Lamp1-Red
    Lamp1 (203,407 20x20), tooltip "If ON, reading is valid.", variable: m_instance.stat.bValid, style: Lamp-Lamp1-Green
    Label (224,406 44x23), "Valid"
    Lamp1 (203,377 20x20), tooltip "pump speed > 0 rpm", variable: m_Instance.stat.bActive, style: Lamp-Lamp1-Blue
    Label (224,376 46x23), "Active"
    Lamp1 (203,495 20x20), tooltip "If ON, reading is valid.", variable: m_instance.stat.bWarningSens_H, style: Lamp-Lamp1-Yellow
    Label (224,494 156x23), "Warning High Sensor"
    Lamp1 (203,465 20x20), tooltip "pump speed > 0 rpm", variable: m_Instance.stat.bWarningSens_HA, style: Lamp-Lamp1-Yellow
    Label (224,464 166x23), "Warning High-Alarm Sensor"
    Lamp1 (203,525 20x20), tooltip "If ON, reading is valid.", variable: m_instance.stat.bWarningSens_L, style: Lamp-Lamp1-Yellow
    Label (224,524 125x23), "Warning Low Sensor"
    Lamp1 (203,552 20x20), tooltip "If ON, reading is valid.", variable: m_instance.stat.bWarningSens_LA, style: Lamp-Lamp1-Yellow
    Label (224,551 164x23), "Warning Low-Alarm Sensor"
    Rectangle (38,593 264x30), "%s", text variable: m_instance.stat.sStatus
    Lamp1 (203,349 20x20), tooltip "pump speed > 0 rpm", variable: m_Instance.stat.bError, style: Lamp-Lamp1-Red
    Label (224,348 46x23), "Error"
    Button (414,19 130x50), "START", input disabled if: m_level_control_instance.bAuto
        OnMouseClick: execute { m_bEnable := TRUE; }
    Button (412,80 130x50), "STOP", input disabled if: m_level_control_instance.bAuto
        OnMouseClick: execute { m_bEnable := FALSE; }
    Rectangle (28,26 334x43), "%s", tooltip "LN2 level control", text variable: m_level_control_instance.in_sName
    Label (329,122 67x23), "LN2 Supply"
    GroupBox (21,659 338x450), "Temperature Thresholds", tooltip "Temp thresholds for LN2 detection and temperature hysteresis"
    GroupBox (38,684 300x200)
    Label (89,701 198x29), "LN2 Detection Temp"
    Textfield (194,748 119x30), "%.1f K", tooltip "LN2 detection temperature threshold", text variable: m_level_control_instance.cfg.lrLN2_Level_SenseTempK_HA, input disabled if: m_level_control_instance.bAuto
        OnMouseClick: write the text variable via Default
    Label (64,749 100x29), "High Alam"
    Textfield (194,778 119x30), "%.1f K", tooltip "LN2 detection temperature threshold", text variable: m_level_control_instance.cfg.lrLN2_Level_SenseTempK_H, input disabled if: m_level_control_instance.bAuto
        OnMouseClick: write the text variable via Default
    Label (64,779 100x29), "High"
    Textfield (194,808 119x30), "%.1f K", tooltip "LN2 detection temperature threshold", text variable: m_level_control_instance.cfg.lrLN2_Level_SenseTempK_L, input disabled if: m_level_control_instance.bAuto
        OnMouseClick: write the text variable via Default
    Label (64,809 100x29), "Low"
    Textfield (194,838 119x30), "%.1f K", tooltip "LN2 detection temperature threshold", text variable: m_level_control_instance.cfg.lrLN2_Level_SenseTempK_LA, input disabled if: m_level_control_instance.bAuto
        OnMouseClick: write the text variable via Default
    Label (64,839 100x29), "Low Alam"
    GroupBox (38,884 300x200)
    Label (89,901 198x29), "LN2 Absent Temp"
    Textfield (194,948 119x30), "%.1f K", tooltip "LN2 detection temperature threshold", text variable: m_level_control_instance.cfg.lrLN2_Level_AbsenceTempK_HA, input disabled if: m_level_control_instance.bAuto
        OnMouseClick: write the text variable via Default
    Label (64,949 100x29), "High Alam"
    Textfield (194,978 119x30), "%.1f K", tooltip "LN2 detection temperature threshold", text variable: m_level_control_instance.cfg.lrLN2_Level_AbsenceTempK_H, input disabled if: m_level_control_instance.bAuto
        OnMouseClick: write the text variable via Default
    Label (64,979 100x29), "High"
    Textfield (194,1008 119x30), "%.1f K", tooltip "LN2 detection temperature threshold", text variable: m_level_control_instance.cfg.lrLN2_Level_AbsenceTempK_L, input disabled if: m_level_control_instance.bAuto
        OnMouseClick: write the text variable via Default
    Label (64,1009 100x29), "Low"
    Textfield (194,1038 119x30), "%.1f K", tooltip "LN2 detection temperature threshold", text variable: m_level_control_instance.cfg.lrLN2_Level_AbsenceTempK_LA, input disabled if: m_level_control_instance.bAuto
        OnMouseClick: write the text variable via Default
    Label (64,1039 100x29), "Low Alam"
    Lamp1 (405,1027 25x25), tooltip "Command coming from the Control System", variable: m_level_control_instance.ctrl.bReadConfig, style: Lamp-Lamp1-Blue
    Button (445,1067 201x31), "Save Configuration", input disabled if: m_level_control_instance.bAuto
        OnMouseClick: execute { m_level_control_instance.ctrl.bWriteConfig := TRUE; }
    Button (445,1027 201x26), "Load Configuration", input disabled if: m_level_control_instance.bAuto
        OnMouseClick: execute { m_level_control_instance.ctrl.bReadConfig := TRUE; }
    Lamp1 (405,1067 25x25), tooltip "Command coming from the Control System", variable: m_level_control_instance.ctrl.bWriteConfig, style: Lamp-Lamp1-Blue
    Rectangle (655,1027 121x30), "%s", text variable: m_level_control_instance.fbConfig.sReadError, colour toggle: m_level_control_instance.fbConfig.bReadError
    Rectangle (655,1067 121x30), "%s", text variable: m_level_control_instance.fbConfig.sWriteError, colour toggle: m_level_control_instance.fbConfig.bWriteError
    Label (329,147 72x23), "LN2 Filling"
END_VISUALIZATION

// HMI/VISUs/Templates/TEMPLATE_MAIN_FSM
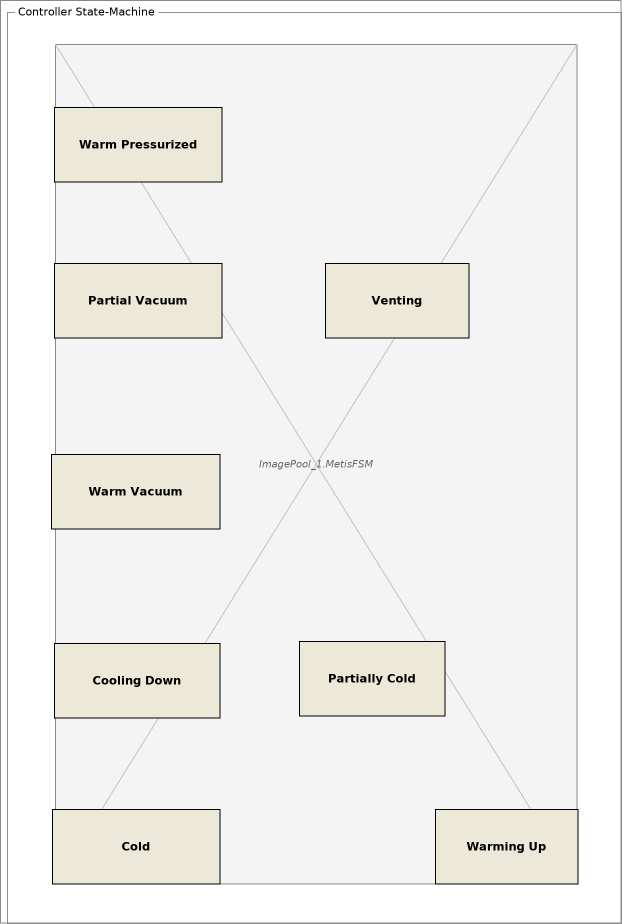
VISUALIZATION TEMPLATE_MAIN_FSM  // 622x924
VAR_IN_OUT
	m_instance:	FB_METIS_CRYO_CTRL;
END_VAR
    GroupBox (7,4 615x920), "Controller State-Machine"
    Group (51,44 527x840)
        Image (4,0 522x840), image: ImagePool_1.MetisFSM
        RoundedRectangle (1,765 168x75), "Cold", colour toggle: m_instance.stat.nState = E_METIS_CRYO_CTRL_STATE.COLD
        RoundedRectangle (3,599 166x75), "Cooling Down", colour toggle: m_instance.stat.nState = E_METIS_CRYO_CTRL_STATE.COOLING_DOWN
        RoundedRectangle (384,765 143x75), "Warming Up", colour toggle: m_instance.stat.nState = E_METIS_CRYO_CTRL_STATE.WARMING_UP
        RoundedRectangle (274,219 144x75), "Venting", colour toggle: m_instance.stat.nState = E_METIS_CRYO_CTRL_STATE.VENTING
        RoundedRectangle (0,410 169x75), "Warm Vacuum", colour toggle: m_instance.stat.nState = E_METIS_CRYO_CTRL_STATE.WARM_VACUUM
        RoundedRectangle (3,63 168x75), "Warm Pressurized", colour toggle: m_instance.stat.nState = E_METIS_CRYO_CTRL_STATE.WARM_PRESS
        RoundedRectangle (3,219 168x75), "Partial Vacuum", colour toggle: m_instance.stat.nState = E_METIS_CRYO_CTRL_STATE.PARTIAL_VACUUM
        RoundedRectangle (248,597 146x75), "Partially Cold", colour toggle: m_instance.stat.nState = E_METIS_CRYO_CTRL_STATE.PARTIALLY_COLD
END_VISUALIZATION

// HMI/VISUs/Templates/TEMPLATE_METIS_CMD_OVERRIDE
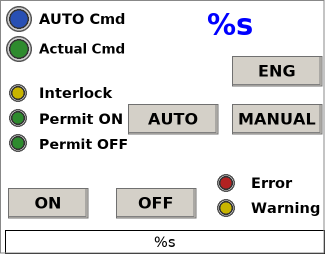
VISUALIZATION TEMPLATE_METIS_CMD_OVERRIDE  // 325x254
VAR_IN_OUT
	m_Cmd:		FB_CRYO_CMD_OVERRIDE;
END_VAR
    Lamp1 (8,83 20x20), variable: m_Cmd.out_bInterlock, style: Lamp-Lamp1-Yellow
    Lamp1 (8,108 20x20), variable: m_Cmd.bPermitOn, style: Lamp-Lamp1-Green
    Lamp1 (8,133 20x20), variable: m_Cmd.bPermitOff, style: Lamp-Lamp1-Green
    Rectangle (36,78 90x30), "Interlock"
    Rectangle (36,104 90x30), "Permit ON"
    Rectangle (36,129 90x30), "Permit OFF"
    Button (8,188 80x30), "ON", colour toggle: (m_Cmd.bPermitOn AND NOT m_Cmd.bAutoMode) OR m_Cmd.bEngMode, input disabled if: m_Cmd.bDisableBtnOn
        OnMouseClick: execute { m_Cmd.bManualCmd := TRUE; }
    Lamp1 (4,34 30x30), tooltip "Actual command going out", variable: m_Cmd.out_bEnable, style: Lamp-Lamp1-Green
    Rectangle (36,34 90x30), "Actual Cmd"
    Button (128,104 90x30), "AUTO", tooltip "Switch to AUTO Mode", colour toggle: m_Cmd.bAutoMode, input disabled if: m_Cmd.bAutoMode OR m_Cmd.bEngMode
        OnMouseClick: execute { m_Cmd.bAutoMode := TRUE; }
    Button (232,104 90x30), "MANUAL", tooltip "Switch to MANUAL Mode", colour toggle: NOT m_Cmd.bAutoMode, input disabled if: NOT m_Cmd.bAutoMode AND NOT m_Cmd.bEngMode
        OnMouseClick: execute { m_Cmd.bAutoMode := FALSE; }
    Button (116,188 80x30), "OFF", colour toggle: (m_Cmd.bPermitOff AND NOT m_Cmd.bAutoMode) OR m_Cmd.bEngMode, input disabled if: m_Cmd.bDisableBtnOff
        OnMouseClick: execute { m_Cmd.bManualCmd := FALSE; }
    Button (232,56 90x30), "ENG", tooltip "Toggle Engineering Mode", colour toggle: m_Cmd.bEngMode, input disabled if: m_Cmd.bAutoMode
        toggle m_Cmd.bEngMode
    Lamp1 (4,4 30x30), tooltip "Command coming from the Control System", variable: m_Cmd.in_bEnable, style: Lamp-Lamp1-Blue
    Rectangle (36,4 90x30), "AUTO Cmd"
    Rectangle (5,230 320x24), "%s", text variable: m_Cmd.out_sStatus
    Lamp1 (216,173 20x20), tooltip "If ON, there is an error in the SW implementation of permission handling.", variable: m_Cmd.out_bError, style: Lamp-Lamp1-Red
    Rectangle (248,168 75x30), "Error"
    Lamp1 (216,198 20x20), tooltip "If ON, ENG command is not safe!", variable: m_Cmd.out_bWarning, style: Lamp-Lamp1-Yellow
    Rectangle (248,193 75x30), "Warning"
    Rectangle (144,4 173x41), "%s", text variable: m_Cmd.out_sMode
END_VISUALIZATION

// HMI/VISUs/Templates/TEMPLATE_METIS_CONTROL_VALVE
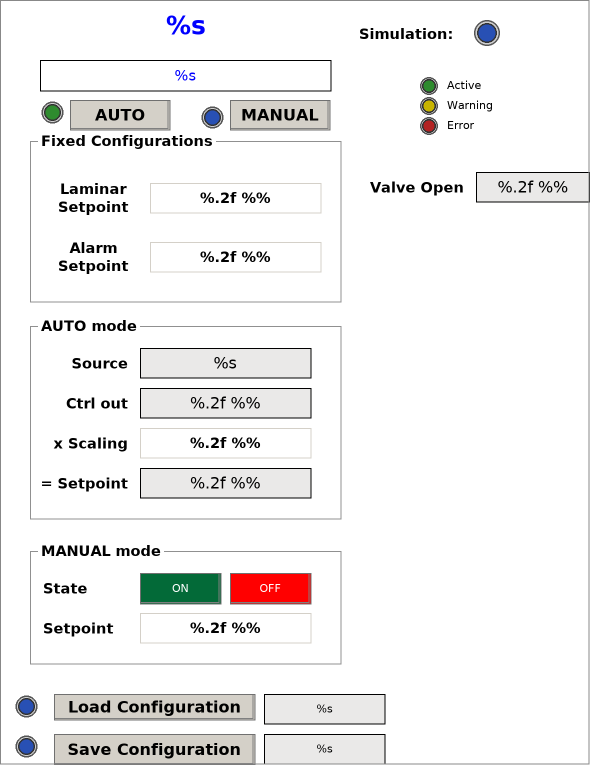
VISUALIZATION TEMPLATE_METIS_CONTROL_VALVE  // 590x765
VAR_IN_OUT
	m_instance: FB_METIS_CONTROL_VALVE;
END_VAR
    GroupBox (30,133 311x169), "Fixed Configurations", tooltip "These configurations are used when no PID control is available."
        Rectangle (18,40 91x50), "Laminar Setpoint", tooltip "Setpoint to achieve laminar flow during normal operations."
        Rectangle (18,99 91x50), "Alarm Setpoint", tooltip "Setpoint during alarm conditions"
    Rectangle (21,10 330x30), "%s", text variable: m_Instance.in_sName
    Group (419,74 112x63)
        Lamp1 (0,2 20x20), tooltip "If ON, Heater is active", variable: m_Instance.stat.bActive, style: Lamp-Lamp1-Green
        Lamp1 (0,22 20x20), tooltip "If ON, reading is in Warning", variable: m_Instance.stat.bWarning, style: Lamp-Lamp1-Yellow
        Lamp1 (0,42 20x20), tooltip "If ON, reading is in error.", variable: m_Instance.stat.bError, style: Lamp-Lamp1-Red
        Label (25,0 87x23), "Active"
        Label (25,20 87x23), "Warning"
        Label (25,40 87x23), "Error"
    Rectangle (476,172 114x30), "%.2f %%", tooltip "Valve open (0 - 100)%", text variable: m_instance.stat.lrActValveFlow
    Lamp1 (472,18 30x30), tooltip "If ON, Heater is simulated.", variable: m_instance.stat.bSimulated, style: Lamp-Lamp1-Blue
    Rectangle (356,19 110x30), "Simulation:"
    Rectangle (356,172 111x31), "Valve Open"
    GroupBox (30,543 311x121), "MANUAL mode"
        Rectangle (10,30 131x31), "State"
        Rectangle (10,70 101x31), "Setpoint"
        Button (110,30 81x31), "ON", input disabled if: NOT m_instance.stat.bManual
            OnMouseClick: execute { m_instance.ctrl.bManualEnable := TRUE; }
        Button (200,30 81x31), "OFF", input disabled if: NOT m_instance.stat.bManual
            OnMouseClick: execute { m_instance.ctrl.bManualEnable := FALSE; }
        Textfield (110,70 171x30), "%.2f %%", text variable: m_instance.ctrl.lrManualSetpoint, input disabled if: NOT m_instance.stat.bManual
            OnMouseClick: write the text variable via Default
    Lamp1 (200,105 25x25), variable: m_instance.stat.bManual, style: Lamp-Lamp1-Blue
    Lamp1 (40,100 25x25), variable: m_instance.stat.bAuto, style: Lamp-Lamp1-Green
    Button (70,100 100x30), "AUTO", tooltip "Switch to AUTO Mode", input disabled if: NOT m_instance.stat.bAcceptCtrlMode_Auto
        OnMouseClick: execute { m_instance.ctrl.eCtrlMode := E_METIS_CTRL_MODE.AUTO; }
    Button (230,100 100x30), "MANUAL", tooltip "Switch to MANUAL Mode", input disabled if: NOT m_instance.stat.bAcceptCtrlMode_Manual
        OnMouseClick: execute { m_instance.ctrl.eCtrlMode := E_METIS_CTRL_MODE.MANUAL; }
    Rectangle (40,60 291x31), "%s", text variable: m_Instance.stat.sValveState
    Lamp1 (14,694 25x25), tooltip "Command coming from the Control System", variable: m_instance.ctrl.bReadConfig, style: Lamp-Lamp1-Blue
    Button (54,734 201x31), "Save Configuration"
        OnMouseClick: execute { m_instance.ctrl.bWriteConfig := TRUE; }
    Button (54,694 201x26), "Load Configuration"
        OnMouseClick: execute { m_instance.ctrl.bReadConfig := TRUE; }
    Lamp1 (14,734 25x25), tooltip "Command coming from the Control System", variable: m_instance.ctrl.bWriteConfig, style: Lamp-Lamp1-Blue
    Rectangle (264,694 121x30), "%s", text variable: m_Instance.fbConfig.sReadError, colour toggle: m_Instance.fbConfig.bReadError
    Rectangle (264,734 121x30), "%s", text variable: m_Instance.fbConfig.sWriteError, colour toggle: m_Instance.fbConfig.bWriteError
    GroupBox (30,318 311x201), "AUTO mode"
        Rectangle (110,30 171x30), "%s", tooltip "Value used by the system [C]", text variable: m_instance.stat.sAutoSetpointSource
        Rectangle (10,30 91x31), "Source"
        Rectangle (10,150 91x31), "= Setpoint", tooltip "Setpoint after the scaling was applied"
        Rectangle (110,150 171x30), "%.2f %%", tooltip "Value used by the system [C]", text variable: m_instance.stat.lrAutoSetpointValue
        Textfield (110,110 171x30), "%.2f %%", text variable: m_instance.cfg.lrAutoScalePercent
            OnMouseClick: write the text variable via Default
        Rectangle (10,110 91x31), "x Scaling", tooltip "Setpoint = controller output x scaling"
        Rectangle (110,70 171x30), "%.2f %%", tooltip "Value used by the system [C]", text variable: m_instance.stat.lrAutoCtrlOut
        Rectangle (10,70 91x31), "Ctrl out", tooltip "Setpoint = controller output x scaling"
    Textfield (150,183 171x30), "%.2f %%", text variable: m_instance.cfg.lrBlowerNormalSetPoint
        OnMouseClick: write the text variable via Default
    Textfield (150,242 171x30), "%.2f %%", text variable: m_instance.cfg.lrBlowerAlarmSetPoint
        OnMouseClick: write the text variable via Default
END_VISUALIZATION

// HMI/VISUs/Templates/TEMPLATE_METIS_CRYO_CPA
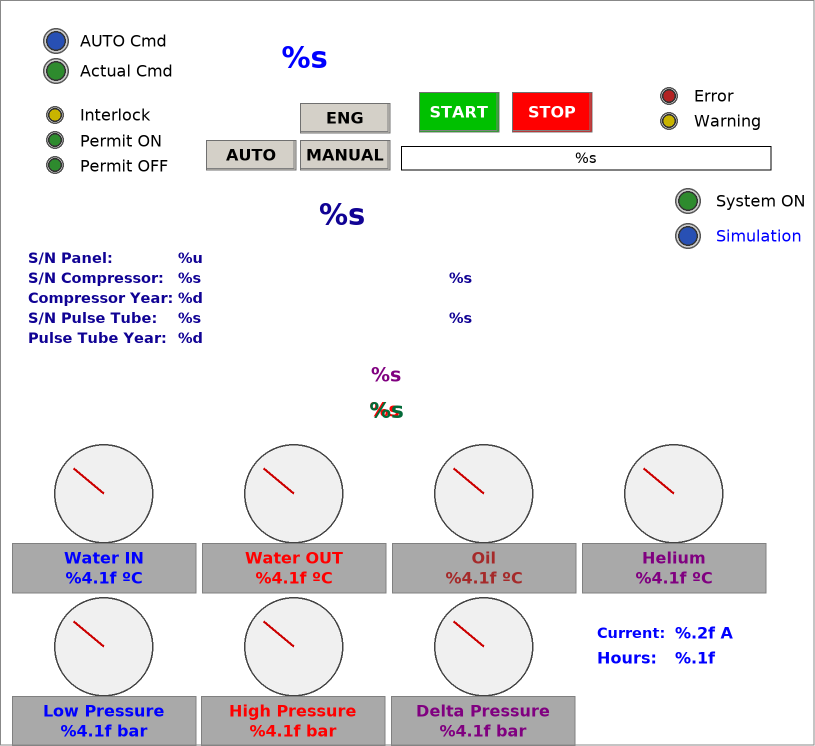
VISUALIZATION TEMPLATE_METIS_CRYO_CPA  // 815x746
VAR_IN_OUT
	m_Instance:	FB_METIS_CRYO_CPA;
	m_Cmd:		FB_CRYO_CMD_OVERRIDE;
END_VAR
    Rectangle (28,197 629x35), "%s", text variable: m_Instance.in_sName
    Rectangle (10,394 750x30), "%s", text variable: m_Instance.stat.sError, invisible if: (m_Instance.stat.nStatusCode<>2)
    Meter180 (4,597 199x99), value: m_Instance.stat.lrLowPressure, style: Meter-Meter180-Gray, scale format: %.0f, scale 0..30
    Rectangle (12,696 184x50), "Low Pressure %4.1f bar", text variable: m_Instance.stat.lrLowPressure
    Meter180 (194,597 199x99), value: m_Instance.stat.lrHighPressure, style: Meter-Meter180-Gray, scale format: %.0f, scale 0..30
    Rectangle (201,696 184x50), "High Pressure %4.1f bar", text variable: m_Instance.stat.lrHighPressure
    Rectangle (10,395 750x30), "%s", text variable: m_Instance.stat.sAlarm, invisible if: (m_Instance.stat.nStatusCode<>1)
    Rectangle (233,394 308x33), "%s", text variable: m_Instance.stat.sStatusOK, invisible if: (m_Instance.stat.nStatusCode<>0 or m_Instance.stat.nOperatingState <>3)
    Meter180 (4,444 199x99), value: m_Instance.stat.lrCoolantInTemp, style: Meter-Meter180-Gray, scale format: %.0f, scale 0..60
    Rectangle (12,543 184x50), "Water IN %4.1f ºC", text variable: m_Instance.stat.lrCoolantInTemp
    Meter180 (194,444 199x99), value: m_Instance.stat.lrCoolantOutTemp, style: Meter-Meter180-Gray, scale format: %.0f, scale 0..60
    Rectangle (202,543 184x50), "Water OUT %4.1f ºC", text variable: m_Instance.stat.lrCoolantOutTemp
    Meter180 (384,444 199x99), value: m_Instance.stat.lrOilTemp, style: Meter-Meter180-Gray, scale format: %.0f, scale 0..60
    Rectangle (392,543 184x50), "Oil %4.1f ºC", text variable: m_Instance.stat.lrOilTemp
    Meter180 (574,444 199x99), value: m_Instance.stat.lrHeliumTemp, style: Meter-Meter180-Gray, scale format: %.0f, scale 0..100
    Rectangle (582,543 184x50), "Helium %4.1f ºC", text variable: m_Instance.stat.lrHeliumTemp
    Rectangle (672,618 95x30), "%.2f A", text variable: m_Instance.stat.lrMotorCurrent
    Rectangle (672,643 95x30), "%.1f", text variable: m_Instance.stat.lrHoursOfOperation
    Rectangle (140,360 493x30), "%s", tooltip "Operational State", text variable: m_Instance.stat.sOperatingState
    Rectangle (175,247 231x22), "%u", text variable: m_Instance.stat.nPanelSerialNumber
    Rectangle (175,267 270x22), "%s", text variable: m_Instance.in_sSN_Compressor
    Rectangle (175,307 270x22), "%s", text variable: m_Instance.in_sSN_PulseTube
    Label (25,247 145x22), "S/N Panel:"
    Label (25,267 145x22), "S/N Compressor:"
    Label (25,307 145x22), "S/N Pulse Tube:"
    Rectangle (594,618 75x30), "Current:"
    Rectangle (594,643 75x30), "Hours:"
    Meter180 (384,597 199x99), value: m_Instance.stat.lrDeltaPressureAverage, style: Meter-Meter180-Gray, scale format: %.0f, scale 0..30
    Rectangle (391,696 184x50), "Delta Pressure %4.1f bar", text variable: m_Instance.stat.lrDeltaPressureAverage
    Label (25,327 145x22), "Pulse Tube Year:"
    Rectangle (175,327 90x22), "%d", text variable: m_Instance.in_nYear_PulseTube
    Label (25,287 145x22), "Compressor Year:"
    Rectangle (175,287 90x22), "%d", text variable: m_Instance.in_nYear_Compressor
    Rectangle (446,267 270x22), "%s", text variable: m_Instance.stat.sServiceDue_Compressor, invisible if: m_Instance.stat.bServiceDue_Compressor=FALSE
        p55702900: m_Instance.stat.wColour_Compressor
    Rectangle (446,307 270x22), "%s", text variable: m_Instance.stat.sServiceDue_PulseTube, invisible if: m_Instance.stat.bServiceDue_PulseTube=FALSE
        p55702900: m_Instance.stat.wColour_PulseTube
    Lamp1 (45,105 20x20), variable: m_Cmd.out_bInterlock, style: Lamp-Lamp1-Yellow
    Lamp1 (45,130 20x20), variable: m_Cmd.bPermitOn, style: Lamp-Lamp1-Green
    Lamp1 (45,155 20x20), variable: m_Cmd.bPermitOff, style: Lamp-Lamp1-Green
    Rectangle (77,100 110x30), "Interlock"
    Rectangle (77,126 110x30), "Permit ON"
    Rectangle (77,151 110x30), "Permit OFF"
    Button (419,92 80x40), "START", colour toggle: (m_Cmd.bPermitOn AND NOT m_Cmd.bAutoMode) OR m_Cmd.bEngMode, input disabled if: m_Cmd.bDisableBtnOn
        OnMouseClick: execute { m_Cmd.bManualCmd := TRUE; }
    Lamp1 (41,56 30x30), tooltip "Actual command going out", variable: m_Cmd.out_bEnable, style: Lamp-Lamp1-Green
    Rectangle (77,56 110x30), "Actual Cmd"
    Button (206,140 90x30), "AUTO", tooltip "Switch to AUTO Mode", colour toggle: m_Cmd.bAutoMode, input disabled if: m_Cmd.bAutoMode OR m_Cmd.bEngMode
        OnMouseClick: execute { m_Cmd.bAutoMode := TRUE; }
    Button (300,140 90x30), "MANUAL", tooltip "Switch to MANUAL Mode", colour toggle: NOT m_Cmd.bAutoMode, input disabled if: NOT m_Cmd.bAutoMode AND NOT m_Cmd.bEngMode
        OnMouseClick: execute { m_Cmd.bAutoMode := FALSE; }
    Button (512,92 80x40), "STOP", colour toggle: (m_Cmd.bPermitOff AND NOT m_Cmd.bAutoMode) OR m_Cmd.bEngMode, input disabled if: m_Cmd.bDisableBtnOff
        OnMouseClick: execute { m_Cmd.bManualCmd := FALSE; }
    Button (300,103 90x30), "ENG", tooltip "Toggle Engineering Mode", colour toggle: m_Cmd.bEngMode, input disabled if: m_Cmd.bAutoMode
        toggle m_Cmd.bEngMode
    Lamp1 (41,26 30x30), tooltip "Command coming from the Control System", variable: m_Cmd.in_bEnable, style: Lamp-Lamp1-Blue
    Rectangle (77,26 110x30), "AUTO Cmd"
    Rectangle (401,146 370x24), "%s", text variable: m_Cmd.out_sStatus
    Lamp1 (659,86 20x20), tooltip "If ON, there is an error in the SW implementation of permission handling.", variable: m_Cmd.out_bError, style: Lamp-Lamp1-Red
    Rectangle (691,81 75x30), "Error"
    Lamp1 (659,111 20x20), tooltip "If ON, ENG command is not safe!", variable: m_Cmd.out_bWarning, style: Lamp-Lamp1-Yellow
    Rectangle (691,106 75x30), "Warning"
    Rectangle (230,37 150x41), "%s", text variable: m_Cmd.out_sMode
    Group (673,221 136x30)
        Lamp1 (0,0 30x30), tooltip "If ON, compressor is simulated", variable: m_Instance.stat.bSimulation, invisible if: NOT m_Instance.stat.bSimulation, style: Lamp-Lamp1-Blue
        Rectangle (40,0 96x30), "Simulation", invisible if: NOT m_Instance.stat.bSimulation
    Group (673,186 142x30)
        Lamp1 (0,0 30x30), tooltip "If ON, compressor is running", variable: m_Instance.stat.bSystemOn, style: Lamp-Lamp1-Green
        Rectangle (40,0 102x30), "System ON", tooltip "Compressor is running"
END_VISUALIZATION

// HMI/VISUs/Templates/TEMPLATE_METIS_CRYO_CPAU60_PID_CTRL
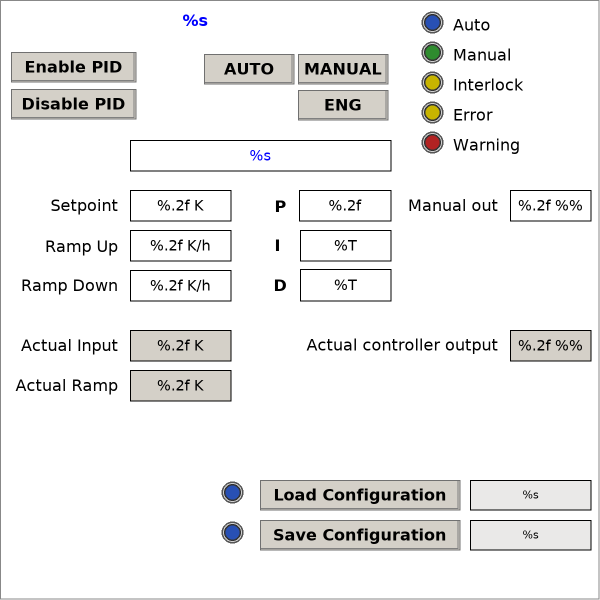
VISUALIZATION TEMPLATE_METIS_CRYO_CPAU60_PID_CTRL  // 600x600
VAR_IN_OUT
	//m_instance	: 	FB_METIS_CTRL_BASE;
	m_instance		:	FB_CPAU60_PID_CTRL;
END_VAR
    Label (450,70 90x30), "Interlock"
    Label (10,330 111x31), "Actual Input"
    Label (30,190 91x31), "Setpoint"
    Rectangle (130,190 101x31), "%.2f K", tooltip "Set point", text variable: m_instance.ctrl.lrManualSetPoint, input disabled if: NOT m_instance.bManualMode AND NOT m_instance.bEngMode
        OnMouseClick: write the text variable via Default
    Rectangle (299,190 92x31), "%.2f", tooltip "Set Velocity [UU/s]", text variable: m_instance.cfg.lrKp, input disabled if: NOT m_instance.bEngMode
        OnMouseClick: write the text variable via Default
    Label (450,100 90x30), "Error"
    Label (450,130 91x30), "Warning"
    Rectangle (510,330 81x31), "%.2f %%", tooltip "Set Velocity [UU/s]", text variable: m_instance.lrControllerOut
    Rectangle (130,330 101x31), "%.2f K", tooltip "Actual Position [UU]", text variable: m_instance.lrActualValue
    Label (10,370 111x31), "Actual Ramp"
    Rectangle (130,370 101x31), "%.2f K", tooltip "Actual Position [UU]", text variable: m_instance.temperature.stat.lrRamp
    Rectangle (300,230 91x31), "%T", tooltip "Set Velocity [UU/s]", text variable: m_instance.cfg.tTn, input disabled if: NOT m_instance.bEngMode
        OnMouseClick: write the text variable via Default
    Rectangle (300,269 91x32), "%T", tooltip "Derivative action time", text variable: m_instance.cfg.tTv, input disabled if: NOT m_instance.bEngMode
        OnMouseClick: write the text variable via Default
    Label (270,190 21x33), "P"
    Label (270,230 21x31), "I"
    Label (270,270 21x31), "D"
    Lamp1 (420,70 25x25), style: Lamp-Lamp1-Yellow
    Lamp1 (420,40 25x25), tooltip "Actual command going out", variable: m_instance.bEngMode, style: Lamp-Lamp1-Green
    Button (11,52 125x30), "Enable PID", tooltip "PID in active mode", colour toggle: m_instance.stat.bEnabled
        OnMouseClick: execute { m_Instance.ctrl.bEnable := TRUE; }
    Lamp1 (420,10 25x25), tooltip "Command coming from the Control System", variable: m_instance.stat.bEnabled, style: Lamp-Lamp1-Blue
    Lamp1 (420,130 25x25), tooltip "If ON, there is an error in the SW implementation of permission handling.", style: Lamp-Lamp1-Red
    Lamp1 (420,100 25x25), tooltip "If ON, ENG command is not safe!", style: Lamp-Lamp1-Yellow
    Rectangle (3,3 385x35), "%s", text variable: m_instance.in_sName
    Label (290,330 211x30), "Actual controller output"
    Rectangle (130,230 101x31), "%.2f K/h", tooltip "Set Velocity [UU/s]", text variable: m_instance.ctrl.lrManualRampUpRate, input disabled if: NOT m_instance.bEngMode
        OnMouseClick: write the text variable via Default
    Label (20,230 101x33), "Ramp Up"
    Button (260,520 200x30), "Save Configuration", input disabled if: NOT m_instance.bEngMode
        OnMouseClick: execute { m_instance.bWriteConfig := TRUE; }
    Button (260,480 200x30), "Load Configuration", input disabled if: NOT m_instance.bEngMode
        OnMouseClick: execute { m_instance.bReadConfig := TRUE; }
    Button (11,89 125x30), "Disable PID", tooltip "PID in Manual mode", colour toggle: NOT m_instance.stat.bEnabled
        OnMouseClick: execute { m_Instance.ctrl.bEnable := FALSE; }
    Label (10,270 111x31), "Ramp Down"
    Rectangle (130,270 101x31), "%.2f K/h", tooltip "Set Velocity [UU/s]", text variable: m_instance.ctrl.lrManualRampDownRate, input disabled if: NOT m_instance.bEngMode
        OnMouseClick: write the text variable via Default
    Button (298,90 90x30), "ENG", tooltip "Toggle Engineering Mode", colour toggle: m_instance.bEngMode, input disabled if: m_instance.bAutoMode
        toggle m_instance.bEngMode
    Button (204,54 90x30), "AUTO", tooltip "Switch to AUTO Mode", colour toggle: m_instance.bAutoMode, input disabled if: m_instance.bAutoMode OR m_instance.bEngMode
        OnMouseClick: execute { m_instance.bAutoMode := TRUE; }
    Button (298,54 90x30), "MANUAL", tooltip "Switch to MANUAL Mode", colour toggle: NOT m_instance.bAutoMode, input disabled if: NOT m_instance.bAutoMode AND NOT m_instance.bEngMode
        OnMouseClick: execute { m_instance.bAutoMode := FALSE; m_instance.bManualMode := TRUE; }
    Rectangle (130,140 261x31), "%s", text variable: m_instance.stat.sStatus
    Rectangle (510,190 81x31), "%.2f %%", tooltip "Set Velocity [UU/s]", text variable: m_instance.lrManualOut, input disabled if: NOT m_instance.bEngMode
        OnMouseClick: write the text variable via Default
    Label (400,190 101x31), "Manual out"
    Lamp1 (220,480 25x25), tooltip "Command coming from the Control System", variable: m_instance.fbTcConfig.bReading, style: Lamp-Lamp1-Blue
    Lamp1 (220,520 25x25), tooltip "Command coming from the Control System", variable: m_instance.fbTcConfig.bWriting, style: Lamp-Lamp1-Blue
    Rectangle (470,480 121x30), "%s", text variable: m_Instance.fbTcConfig.nReadErrorCode, colour toggle: m_Instance.fbTcConfig.bReadError
    Rectangle (470,520 121x30), "%s", text variable: m_Instance.fbTcConfig.sWriteError, colour toggle: m_Instance.fbTcConfig.bWriteError
    Label (450,40 90x30), "Manual"
    Label (450,10 111x30), "Auto"
END_VISUALIZATION

// HMI/VISUs/Templates/TEMPLATE_METIS_CRYO_PWM_PID_CTRL
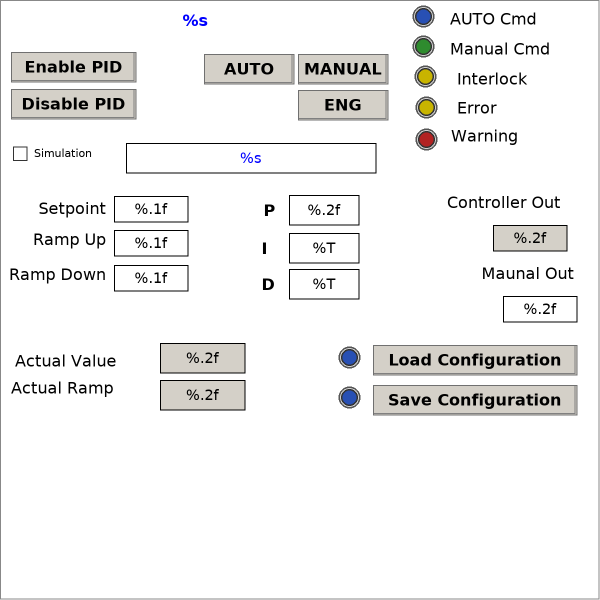
VISUALIZATION TEMPLATE_METIS_CRYO_PWM_PID_CTRL  // 600x600
VAR_IN_OUT
	//m_instance	: 	FB_METIS_CTRL_BASE;
	m_instance		:	FB_PWM_PID_CTRL;
	m_bEnable	:	BOOL;
	
END_VAR
    Label (454,64 90x30), "Interlock"
    Label (12,346 151x30), "Actual Value"
    Label (37,197 72x23), "Setpoint"
    Rectangle (114,196 74x26), "%.1f", tooltip "Set point", text variable: m_instance.ctrl.lrManualSetPoint, input disabled if: NOT m_instance.bManualMode AND NOT m_instance.bEngMode
        OnMouseClick: write the text variable via Default
    Rectangle (289,195 70x30), "%.2f", tooltip "Set Velocity [UU/s]", text variable: m_instance.cfg.lrKp, input disabled if: NOT m_instance.bEngMode
        OnMouseClick: write the text variable via Default
    Label (454,93 90x30), "Error"
    Label (448,121 91x30), "Warning"
    Rectangle (493,225 74x26), "%.2f", tooltip "Set Velocity [UU/s]", text variable: m_instance.lrControllerOut
    Rectangle (160,343 85x30), "%.2f", tooltip "Actual Position [UU]", text variable: m_instance.lrActualValue
    Label (8,373 118x30), "Actual Ramp"
    Rectangle (160,380 85x30), "%.2f", tooltip "Actual Position [UU]", text variable: m_instance.temperature.stat.lrRamp
    Rectangle (289,233 70x30), "%T", tooltip "Set Velocity [UU/s]", text variable: m_instance.cfg.tTn, input disabled if: NOT m_instance.bEngMode
        OnMouseClick: write the text variable via Default
    Rectangle (289,269 70x30), "%T", tooltip "Derivative action time", text variable: m_instance.cfg.tTv, input disabled if: NOT m_instance.bEngMode
        OnMouseClick: write the text variable via Default
    Label (258,198 20x25), "P"
    Label (261,236 15x25), "I"
    Label (258,272 20x25), "D"
    Lamp1 (413,64 25x25), style: Lamp-Lamp1-Yellow
    Lamp1 (411,34 25x25), tooltip "Actual command going out", variable: m_instance.bEngMode, style: Lamp-Lamp1-Green
    Rectangle (447,34 110x30), "Manual Cmd"
    Button (11,52 125x30), "Enable PID", tooltip "PID in active mode", colour toggle: m_instance.stat.bEnabled
        OnMouseClick: execute { m_bEnable := TRUE; }
    Lamp1 (411,4 25x25), tooltip "Command coming from the Control System", variable: m_instance.stat.bEnabled, style: Lamp-Lamp1-Blue
    Rectangle (447,4 110x30), "AUTO Cmd"
    Lamp1 (414,127 25x25), tooltip "If ON, there is an error in the SW implementation of permission handling.", style: Lamp-Lamp1-Red
    Lamp1 (414,95 25x25), tooltip "If ON, ENG command is not safe!", style: Lamp-Lamp1-Yellow
    Rectangle (3,3 385x35), "%s"
    Label (444,191 123x23), "Controller Out"
    Rectangle (114,230 74x26), "%.1f", tooltip "Set Velocity [UU/s]", text variable: m_instance.ctrl.lrManualRampUpRate, input disabled if: NOT m_instance.bEngMode
        OnMouseClick: write the text variable via Default
    Label (25,228 84x23), "Ramp Up"
    Checkbox (11,136 123x35), "Simulation", input disabled if: NOT m_instance.bEngMode
    Button (373,385 204x30), "Save Configuration", input disabled if: NOT m_instance.bEngMode
        OnMouseClick: execute { m_instance.bWriteConfig := TRUE; }
    Button (373,345 204x30), "Load Configuration", input disabled if: NOT m_instance.bEngMode
        OnMouseClick: execute { m_instance.bReadConfig := TRUE; }
    Button (11,89 125x30), "Disable PID", tooltip "PID in Manual mode", colour toggle: NOT m_instance.stat.bEnabled
        OnMouseClick: execute { m_bEnable := FALSE; }
    Label (3,263 106x23), "Ramp Down"
    Rectangle (114,265 74x26), "%.1f", tooltip "Set Velocity [UU/s]", text variable: m_instance.ctrl.lrManualRampDownRate, input disabled if: NOT m_instance.bEngMode
        OnMouseClick: write the text variable via Default
    Button (298,90 90x30), "ENG", tooltip "Toggle Engineering Mode", colour toggle: m_instance.bEngMode, input disabled if: m_instance.bAutoMode
        toggle m_instance.bEngMode
    Button (204,54 90x30), "AUTO", tooltip "Switch to AUTO Mode", colour toggle: m_instance.bAutoMode, input disabled if: m_instance.bAutoMode OR m_instance.bEngMode
        OnMouseClick: execute { m_instance.bAutoMode := TRUE; }
    Button (298,54 90x30), "MANUAL", tooltip "Switch to MANUAL Mode", colour toggle: NOT m_instance.bAutoMode, input disabled if: NOT m_instance.bAutoMode AND NOT m_instance.bEngMode
        OnMouseClick: execute { m_instance.bAutoMode := FALSE; m_instance.bManualMode := TRUE; }
    Rectangle (126,143 250x30), "%s", text variable: m_instance.stat.sStatus
    Rectangle (503,296 74x26), "%.2f", tooltip "Set Velocity [UU/s]", text variable: m_instance.lrManualOut, input disabled if: NOT m_instance.bEngMode
        OnMouseClick: write the text variable via Default
    Label (454,262 123x23), "Maunal Out"
    Lamp1 (337,345 25x25), tooltip "Command coming from the Control System", variable: m_instance.bReadConfig, style: Lamp-Lamp1-Blue
    Lamp1 (337,385 25x25), tooltip "Command coming from the Control System", variable: m_instance.bWriteConfig, style: Lamp-Lamp1-Blue
END_VISUALIZATION

// HMI/VISUs/Templates/TEMPLATE_METIS_CTRL_TEMPERATURE
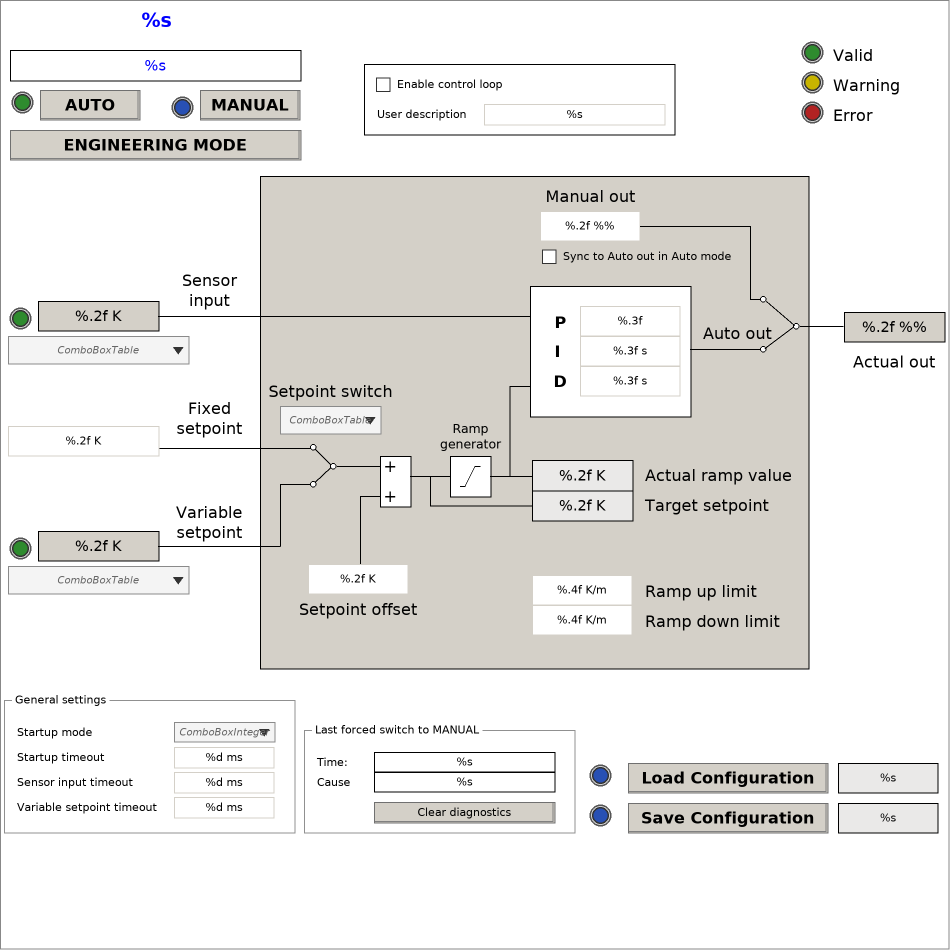
VISUALIZATION TEMPLATE_METIS_CTRL_TEMPERATURE  // 950x950
VAR_IN_OUT
	m_instance  : FB_METIS_CTRL_TEMPERATURE;
    m_temp      : FB_METIS_TEMPERATURES;
END_VAR
    Rectangle (364,64 311x71)
    Rectangle (260,176 549x493)
    Label (172,268 75x45), "Sensor input"
    Label (830,100 90x31), "Error"
    Label (830,70 91x31), "Warning"
    Rectangle (844,312 101x30), "%.2f %%", tooltip "Set Velocity [UU/s]", text variable: m_instance.stat.lrControllerOut
    Rectangle (38,301 121x30), "%.2f K", tooltip "Actual input temperature", text variable: m_instance.stat.lrActInput
    Label (642,490 171x31), "Target setpoint"
    Rectangle (532,490 101x31), "%.2f K", tooltip "Target ramp setpoint", text variable: m_instance.stat.lrTargetSetpoint
    Lamp1 (170,95 25x25), variable: m_instance.stat.bCtrlModeIsManual, style: Lamp-Lamp1-Blue
    Lamp1 (10,90 25x25), variable: m_instance.stat.bCtrlModeIsAuto, style: Lamp-Lamp1-Green
    Lamp1 (800,70 25x25), variable: m_instance.stat.bWarning, style: Lamp-Lamp1-Yellow
    Lamp1 (800,100 25x25), variable: m_instance.stat.bError, style: Lamp-Lamp1-Red
    Rectangle (3,3 308x35), "%s", text variable: m_instance.in_sName
    Label (700,316 81x35), "Auto out"
    Label (642,575 161x33), "Ramp up limit"
    Label (430,416 81x41), "Ramp generator"
    Button (40,90 100x30), "AUTO", tooltip "Switch to AUTO Mode", input disabled if: m_instance.stat.bAcceptCtrlMode_Manual
        OnMouseClick: execute { m_instance.ctrl.eCtrlMode := E_METIS_CTRL_MODE.AUTO; }
    Button (200,90 100x30), "MANUAL", tooltip "Switch to MANUAL Mode", input disabled if: m_instance.stat.bAcceptCtrlMode_Auto
        OnMouseClick: execute { m_instance.ctrl.eCtrlMode := E_METIS_CTRL_MODE.MANUAL; }
    Rectangle (10,50 291x31), "%s", text variable: m_instance.stat.sStatus
    Label (540,181 101x31), "Manual out"
    Button (628,803 200x30), "Save Configuration", input disabled if: NOT m_instance.stat.bEngMode
        OnMouseClick: execute { m_instance.ctrl.bWriteConfig := TRUE; }
    Button (628,763 200x30), "Load Configuration", input disabled if: NOT m_instance.stat.bEngMode
        OnMouseClick: execute { m_instance.ctrl.bReadConfig := TRUE; }
    Lamp1 (588,763 25x25), tooltip "Command coming from the Control System", variable: m_instance.fbTcConfig.bReading, style: Lamp-Lamp1-Blue
    Lamp1 (588,803 25x25), tooltip "Command coming from the Control System", variable: m_instance.fbTcConfig.bWriting, style: Lamp-Lamp1-Blue
    Rectangle (838,763 100x30), "%s", text variable: m_Instance.fbTcConfig.sReadError, colour toggle: m_Instance.fbTcConfig.bReadError
    Rectangle (838,803 100x30), "%s", text variable: m_Instance.fbTcConfig.sWriteError, colour toggle: m_Instance.fbTcConfig.bWriteError
    Line (158,316) (588,316)
    Line (158,448) (312,448)
    ComboBoxTable (8,336 181x28), input disabled if: NOT m_instance.stat.bEngMode, data array: m_temp.all_temperature_names
        p3854506369: m_temp.all_temperature_names[INDEX]
    Label (172,396 75x45), "Fixed setpoint"
    Rectangle (38,531 121x30), "%.2f K", tooltip "Actual variable setpoint temperature", text variable: m_instance.stat.lrActVariableSetpoint
    ComboBoxTable (8,566 181x28), input disabled if: NOT m_instance.stat.bEngMode, data array: m_temp.all_temperature_names
        p3854506369: m_temp.all_temperature_names[INDEX]
    Line (158,546) (280,546)
    Label (172,500 75x45), "Variable setpoint"
    Line (314,448) (330,464), invisible if: NOT m_instance.stat.bSetpointSwitchIsFixed
    Line (337,466) (380,466)
    Label (260,376 141x31), "Setpoint switch"
    Rectangle (380,456 31x51)
    Line (410,476) (450,476)
    Label (380,456 21x21), "+"
    Label (380,486 21x21), "+"
    Line (360,496) (380,496)
    Line (360,496) (360,564)
    Label (288,594 141x31), "Setpoint offset"
    Rectangle (450,456 41x41)
    Line (460,486) (465,486)
    Line (465,486) (475,466)
    Line (475,466) (480,466)
    Line (490,476) (580,476)
    Line (510,476) (510,386)
    Rectangle (530,286 161x131)
    Label (550,306 21x33), "P"
    Label (550,336 21x31), "I"
    Label (550,366 21x31), "D"
    Line (510,386) (530,386)
    Label (642,605 143x33), "Ramp down limit"
    Line (430,476) (430,506)
    Line (690,349) (763,349)
    Line (750,226) (750,299)
    Ellipse (760,346 6x6)
    Ellipse (793,323 6x6)
    Line (800,326) (843,326)
    Line (766,301) (794,325), invisible if: NOT m_instance.stat.bCtrlModeIsManual
    Label (844,347 101x30), "Actual out"
    Ellipse (330,463 6x6)
    Ellipse (310,481 6x6)
    Ellipse (310,444 6x6)
    ComboBoxTable (280,406 101x28), tooltip "Switch between the fixed and the variable setpoint", variable: m_instance.cfg.eSetpointSwitch, input disabled if: NOT m_instance.stat.bEngMode, data array: m_instance.aSetpointSwitchNames
        p3854506369: m_instance.aSetpointSwitchNames[INDEX]
    Line (280,484) (280,546)
    Line (280,484) (310,484)
    Checkbox (374,74 171x21), "Enable control loop", variable: m_Instance.cfg.bEnabled, input disabled if: NOT m_instance.stat.bEngMode
    Label (374,104 101x21), "User description"
    Textfield (484,104 181x21), "%s", text variable: m_Instance.cfg.sDescription, input disabled if: NOT m_instance.stat.bEngMode
        OnMouseClick: write the text variable via Default
    Button (10,130 291x30), "ENGINEERING MODE", tooltip "Toggle Engineering Mode", colour toggle: m_instance.stat.bEngMode, pressed state: m_instance.stat.bEngMode
        toggle m_instance.ctrl.bEngMode
    Line (532,506) (430,506)
    Rectangle (532,460 101x31), "%.2f K", tooltip "Transient ramp setpoint", text variable: m_instance.stat.lrRampValue
    Label (642,460 171x31), "Actual ramp value"
    Textfield (532,575 100x30), "%.4f K/m", tooltip "Max warming up rate", text variable: m_instance.cfg.lrRampUpRate, input disabled if: NOT m_instance.stat.bEngMode
        OnMouseClick: write the text variable via Default
    Textfield (532,605 100x30), "%.4f K/m", tooltip "Max cooldown rate", text variable: m_instance.cfg.lrRampDownRate, input disabled if: NOT m_instance.stat.bEngMode
        OnMouseClick: write the text variable via Default
    Textfield (580,306 100x30), "%.3f", tooltip "Gain (Kp)", text variable: m_instance.cfg.lrKp, input disabled if: NOT m_instance.stat.bEngMode
        OnMouseClick: write the text variable via Default
    Textfield (580,336 100x30), "%.3f s", tooltip "Integral part (Tn)", text variable: m_instance.cfg.lrTn, input disabled if: NOT m_instance.stat.bEngMode
        OnMouseClick: write the text variable via Default
    Textfield (580,366 100x30), "%.3f s", tooltip "Derivative part (Td)", text variable: m_instance.cfg.lrTd, input disabled if: NOT m_instance.stat.bEngMode
        OnMouseClick: write the text variable via Default
    Textfield (308,564 100x30), "%.2f K", tooltip "Offset added to the setpoint (optional, put to 0 if not needed)", text variable: m_instance.ctrl.lrSetpointOffset, input disabled if: NOT m_instance.stat.bEngMode
        OnMouseClick: write the text variable via Default
    Textfield (8,426 151x30), "%.2f K", tooltip "Fixed setpoint temperature", text variable: m_instance.ctrl.lrFixedSetpoint, input disabled if: NOT m_instance.stat.bEngMode
        OnMouseClick: write the text variable via Default
    Line (315,482) (331,467), invisible if: NOT m_instance.stat.bSetpointSwitchIsVariable
    Line (765,348) (793,327), invisible if: NOT m_instance.stat.bCtrlModeIsAuto
    Line (750,299) (763,299)
    Textfield (540,211 100x30), "%.2f %%", tooltip "Manual output percentage", text variable: m_instance.ctrl.lrManualOut, input disabled if: (NOT m_instance.stat.bEngMode) AND (m_instance.stat.bCtrlModeIsAuto)
        OnMouseClick: write the text variable via Default
    Lamp1 (8,306 25x25), tooltip "Green if the input temperature is valid", variable: m_instance.stat.bActInputValid, style: Lamp-Lamp1-Green
    Lamp1 (8,536 25x25), tooltip "Green if the variable setpoint temperature is valid", variable: m_instance.stat.bActVariableSetpointValid, style: Lamp-Lamp1-Green
    Checkbox (540,246 191x21), "Sync to Auto out in Auto mode", tooltip "During AUTO mode, continuously update the manual output", variable: m_instance.cfg.bSyncManualOut, input disabled if: NOT m_instance.stat.bEngMode
    Line (640,226) (750,226)
    Label (830,40 91x31), "Valid"
    Lamp1 (800,40 25x25), variable: m_instance.stat.bValid, style: Lamp-Lamp1-Green
    GroupBox (4,692 291x141), "General settings"
        Textfield (170,55 100x21), "%d ms", tooltip "Maximum time before the input temperature (and if used, the variable setpoint temperature) must be valid. Otherwise the Error flag is set, and the control mode is forced to MANUAL.", text variable: m_instance.cfg.nStartupTimeout, input disabled if: NOT m_instance.stat.bEngMode
            OnMouseClick: write the text variable via Default
        Label (10,55 101x21), "Startup timeout"
        Label (10,30 101x21), "Startup mode"
        ComboBoxInteger (170,30 101x20), variable: m_instance.cfg.eStartupCtrlMode, input disabled if: NOT m_instance.stat.bEngMode, text list: 'TEXTLIST_METIS_CTRL_MODE'
        Label (10,80 121x21), "Sensor input timeout"
        Label (10,105 161x21), "Variable setpoint timeout"
        Textfield (170,80 100x21), "%d ms", tooltip "Maximum time that the input sensor can be invalid, before automatically switching to AUTO.", text variable: m_instance.cfg.nInputTempTimeout, input disabled if: NOT m_instance.stat.bEngMode
            OnMouseClick: write the text variable via Default
        Textfield (170,105 100x21), "%d ms", tooltip "Maximum time that the variable setpoint sensor can be invalid, before automatically switching to AUTO.", text variable: m_instance.cfg.nSetpointTempTimeout, input disabled if: NOT m_instance.stat.bEngMode
            OnMouseClick: write the text variable via Default
    GroupBox (304,722 271x111), "Last forced switch to MANUAL"
        Label (10,30 61x21), "Time:"
        Label (10,50 61x21), "Cause"
        Rectangle (70,30 181x20), "%s", text variable: m_instance.stat.sLastForcedManualTime
        Rectangle (70,50 181x20), "%s", text variable: m_instance.stat.sLastForcedManualCause
        Button (70,80 181x21), "Clear diagnostics", input disabled if: NOT m_instance.stat.bEngMode
            OnMouseClick: execute { m_instance.ctrl.bClearForcedManualDiag := TRUE; }
    Ellipse (760,296 6x6)
END_VISUALIZATION

// HMI/VISUs/Templates/TEMPLATE_METIS_CTRL_TEMPERATURE_MPIA
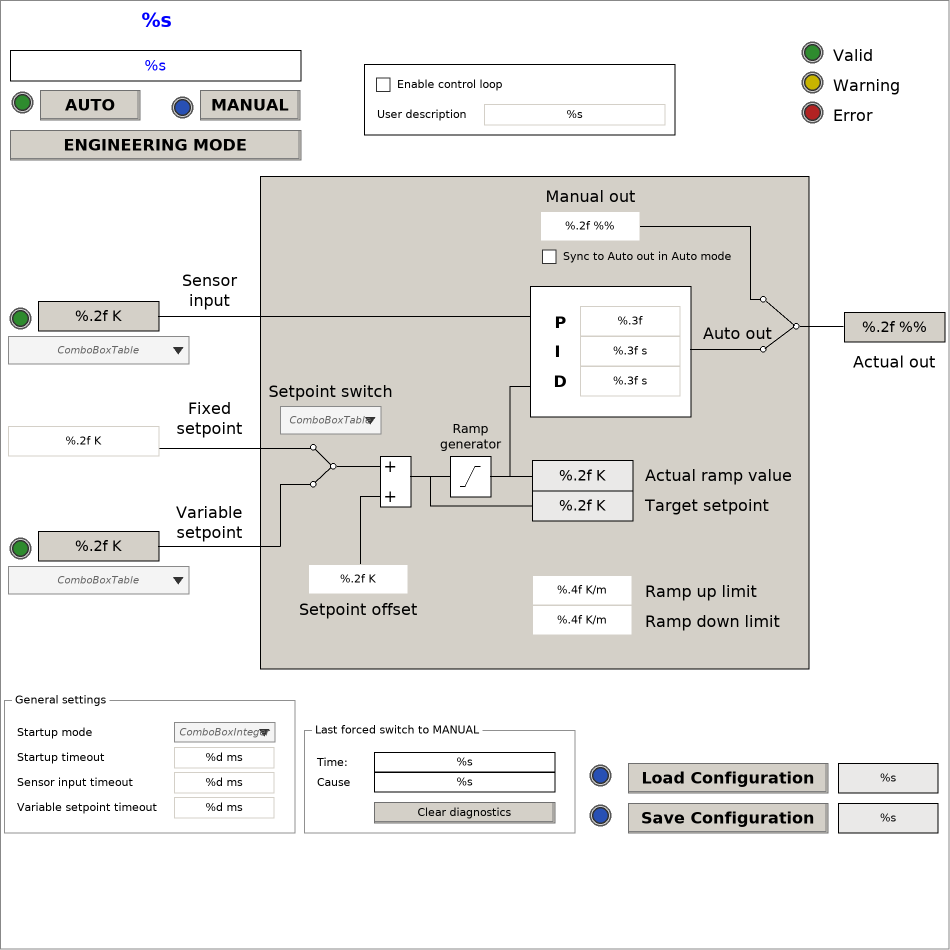
VISUALIZATION TEMPLATE_METIS_CTRL_TEMPERATURE_MPIA  // 950x950
VAR_IN_OUT
	m_instance  : FB_METIS_CTRL_TEMPERATURE;
    m_temp      : FB_METIS_TEMPERATURES;
END_VAR
    Rectangle (364,64 311x71)
    Rectangle (260,176 549x493)
    Label (172,268 75x45), "Sensor input"
    Label (830,100 90x31), "Error"
    Label (830,70 91x31), "Warning"
    Rectangle (844,312 101x30), "%.2f %%", tooltip "Set Velocity [UU/s]", text variable: m_instance.stat.lrControllerOut
    Rectangle (38,301 121x30), "%.2f K", tooltip "Actual input temperature", text variable: m_instance.stat.lrActInput
    Label (642,490 171x31), "Target setpoint"
    Rectangle (532,490 101x31), "%.2f K", tooltip "Target ramp setpoint", text variable: m_instance.stat.lrTargetSetpoint
    Lamp1 (170,95 25x25), variable: m_instance.stat.bCtrlModeIsManual, style: Lamp-Lamp1-Blue
    Lamp1 (10,90 25x25), variable: m_instance.stat.bCtrlModeIsAuto, style: Lamp-Lamp1-Green
    Lamp1 (800,70 25x25), variable: m_instance.stat.bWarning, style: Lamp-Lamp1-Yellow
    Lamp1 (800,100 25x25), variable: m_instance.stat.bError, style: Lamp-Lamp1-Red
    Rectangle (3,3 308x35), "%s", text variable: m_instance.in_sName
    Label (700,316 81x35), "Auto out"
    Label (642,575 161x33), "Ramp up limit"
    Label (430,416 81x41), "Ramp generator"
    Button (40,90 100x30), "AUTO", tooltip "Switch to AUTO Mode", input disabled if: m_instance.stat.bAcceptCtrlMode_Manual
        OnMouseClick: execute { m_instance.ctrl.eCtrlMode := E_METIS_CTRL_MODE.AUTO; }
    Button (200,90 100x30), "MANUAL", tooltip "Switch to MANUAL Mode", input disabled if: m_instance.stat.bAcceptCtrlMode_Auto
        OnMouseClick: execute { m_instance.ctrl.eCtrlMode := E_METIS_CTRL_MODE.MANUAL; }
    Rectangle (10,50 291x31), "%s", text variable: m_instance.stat.sStatus
    Label (540,181 101x31), "Manual out"
    Group (588,763 350x70)
        Button (40,40 200x30), "Save Configuration", input disabled if: NOT m_instance.stat.bEngMode
            OnMouseClick: execute { m_instance.ctrl.bWriteConfig := TRUE; }
        Button (40,0 200x30), "Load Configuration", input disabled if: NOT m_instance.stat.bEngMode
            OnMouseClick: execute { m_instance.ctrl.bReadConfig := TRUE; }
        Lamp1 (0,0 25x25), tooltip "Command coming from the Control System", variable: m_instance.fbTcConfig.bReading, style: Lamp-Lamp1-Blue
        Lamp1 (0,40 25x25), tooltip "Command coming from the Control System", variable: m_instance.fbTcConfig.bWriting, style: Lamp-Lamp1-Blue
        Rectangle (250,0 100x30), "%s", text variable: m_Instance.fbTcConfig.sReadError, colour toggle: m_Instance.fbTcConfig.bReadError
        Rectangle (250,40 100x30), "%s", text variable: m_Instance.fbTcConfig.sWriteError, colour toggle: m_Instance.fbTcConfig.bWriteError
    Line (158,316) (588,316)
    Line (158,448) (312,448)
    ComboBoxTable (8,336 181x28), variable: m_instance.ctrl.nInputTempIndex, input disabled if: NOT m_instance.stat.bEngMode, data array: m_temp.all_temperature_names
        p3854506369: m_temp.all_temperature_names[INDEX]
    Label (172,396 75x45), "Fixed setpoint"
    Rectangle (38,531 121x30), "%.2f K", tooltip "Actual variable setpoint temperature", text variable: m_instance.stat.lrActVariableSetpoint
    ComboBoxTable (8,566 181x28), variable: m_instance.ctrl.nSetpointTempIndex, input disabled if: NOT m_instance.stat.bEngMode, data array: m_temp.all_temperature_names
        p3854506369: m_temp.all_temperature_names[INDEX]
    Line (158,546) (280,546)
    Label (172,500 75x45), "Variable setpoint"
    Line (314,448) (330,464), invisible if: NOT m_instance.stat.bSetpointSwitchIsFixed
    Line (337,466) (380,466)
    Label (260,376 141x31), "Setpoint switch"
    Rectangle (380,456 31x51)
    Line (410,476) (450,476)
    Label (380,456 21x21), "+"
    Label (380,486 21x21), "+"
    Line (360,496) (380,496)
    Line (360,496) (360,564)
    Label (288,594 141x31), "Setpoint offset"
    Rectangle (450,456 41x41)
    Line (460,486) (465,486)
    Line (465,486) (475,466)
    Line (475,466) (480,466)
    Line (490,476) (580,476)
    Line (510,476) (510,386)
    Rectangle (530,286 161x131)
    Label (550,306 21x33), "P"
    Label (550,336 21x31), "I"
    Label (550,366 21x31), "D"
    Line (510,386) (530,386)
    Label (642,605 143x33), "Ramp down limit"
    Line (430,476) (430,506)
    Line (690,349) (763,349)
    Line (750,226) (750,299)
    Ellipse (760,346 6x6)
    Ellipse (793,323 6x6)
    Line (800,326) (843,326)
    Line (766,301) (794,325), invisible if: NOT m_instance.stat.bCtrlModeIsManual
    Label (844,347 101x30), "Actual out"
    Ellipse (330,463 6x6)
    Ellipse (310,481 6x6)
    Ellipse (310,444 6x6)
    ComboBoxTable (280,406 101x28), tooltip "Switch between the fixed and the variable setpoint", variable: m_instance.cfg.eSetpointSwitch, input disabled if: NOT m_instance.stat.bEngMode, data array: m_instance.aSetpointSwitchNames
        p3854506369: m_instance.aSetpointSwitchNames[INDEX]
    Line (280,484) (280,546)
    Line (280,484) (310,484)
    Checkbox (374,74 171x21), "Enable control loop", variable: m_Instance.cfg.bEnabled, input disabled if: NOT m_instance.stat.bEngMode
    Label (374,104 101x21), "User description"
    Textfield (484,104 181x21), "%s", text variable: m_Instance.cfg.sDescription, input disabled if: NOT m_instance.stat.bEngMode
        OnMouseClick: write the text variable via Default
    Button (10,130 291x30), "ENGINEERING MODE", tooltip "Toggle Engineering Mode", colour toggle: m_instance.stat.bEngMode, pressed state: m_instance.stat.bEngMode
        toggle m_instance.ctrl.bEngMode
    Line (532,506) (430,506)
    Rectangle (532,460 101x31), "%.2f K", tooltip "Transient ramp setpoint", text variable: m_instance.stat.lrRampValue
    Label (642,460 171x31), "Actual ramp value"
    Textfield (532,575 100x30), "%.4f K/m", tooltip "Max warming up rate", text variable: m_instance.cfg.lrRampUpRate, input disabled if: NOT m_instance.stat.bEngMode
        OnMouseClick: write the text variable via Default
    Textfield (532,605 100x30), "%.4f K/m", tooltip "Max cooldown rate", text variable: m_instance.cfg.lrRampDownRate, input disabled if: NOT m_instance.stat.bEngMode
        OnMouseClick: write the text variable via Default
    Textfield (580,306 100x30), "%.3f", tooltip "Gain (Kp)", text variable: m_instance.cfg.lrKp, input disabled if: NOT m_instance.stat.bEngMode
        OnMouseClick: write the text variable via Default
    Textfield (580,336 100x30), "%.3f s", tooltip "Integral part (Tn)", text variable: m_instance.cfg.lrTn, input disabled if: NOT m_instance.stat.bEngMode
        OnMouseClick: write the text variable via Default
    Textfield (580,366 100x30), "%.3f s", tooltip "Derivative part (Td)", text variable: m_instance.cfg.lrTd, input disabled if: NOT m_instance.stat.bEngMode
        OnMouseClick: write the text variable via Default
    Textfield (308,564 100x30), "%.2f K", tooltip "Offset added to the setpoint (optional, put to 0 if not needed)", text variable: m_instance.ctrl.lrSetpointOffset, input disabled if: NOT m_instance.stat.bEngMode
        OnMouseClick: write the text variable via Default
    Textfield (8,426 151x30), "%.2f K", tooltip "Fixed setpoint temperature", text variable: m_instance.ctrl.lrFixedSetpoint, input disabled if: NOT m_instance.stat.bEngMode
        OnMouseClick: write the text variable via Default
    Line (315,482) (331,467), invisible if: NOT m_instance.stat.bSetpointSwitchIsVariable
    Line (765,348) (793,327), invisible if: NOT m_instance.stat.bCtrlModeIsAuto
    Line (750,299) (763,299)
    Textfield (540,211 100x30), "%.2f %%", tooltip "Manual output percentage", text variable: m_instance.ctrl.lrManualOut, input disabled if: (NOT m_instance.stat.bEngMode) AND (m_instance.stat.bCtrlModeIsAuto)
        OnMouseClick: write the text variable via Default
    Lamp1 (8,306 25x25), tooltip "Green if the input temperature is valid", variable: m_instance.stat.bActInputValid, style: Lamp-Lamp1-Green
    Lamp1 (8,536 25x25), tooltip "Green if the variable setpoint temperature is valid", variable: m_instance.stat.bActVariableSetpointValid, style: Lamp-Lamp1-Green
    Checkbox (540,246 191x21), "Sync to Auto out in Auto mode", tooltip "During AUTO mode, continuously update the manual output", variable: m_instance.cfg.bSyncManualOut, input disabled if: NOT m_instance.stat.bEngMode
    Line (640,226) (750,226)
    Label (830,40 91x31), "Valid"
    Lamp1 (800,40 25x25), variable: m_instance.stat.bValid, style: Lamp-Lamp1-Green
    GroupBox (4,692 291x141), "General settings"
        Textfield (170,55 100x21), "%d ms", tooltip "Maximum time before the input temperature (and if used, the variable setpoint temperature) must be valid. Otherwise the Error flag is set, and the control mode is forced to MANUAL.", text variable: m_instance.cfg.nStartupTimeout, input disabled if: NOT m_instance.stat.bEngMode
            OnMouseClick: write the text variable via Default
        Label (10,55 101x21), "Startup timeout"
        Label (10,30 101x21), "Startup mode"
        ComboBoxInteger (170,30 101x20), variable: m_instance.cfg.eStartupCtrlMode, input disabled if: NOT m_instance.stat.bEngMode, text list: 'TEXTLIST_METIS_CTRL_MODE'
        Label (10,80 121x21), "Sensor input timeout"
        Label (10,105 161x21), "Variable setpoint timeout"
        Textfield (170,80 100x21), "%d ms", tooltip "Maximum time that the input sensor can be invalid, before automatically switching to AUTO.", text variable: m_instance.cfg.nInputTempTimeout, input disabled if: NOT m_instance.stat.bEngMode
            OnMouseClick: write the text variable via Default
        Textfield (170,105 100x21), "%d ms", tooltip "Maximum time that the variable setpoint sensor can be invalid, before automatically switching to AUTO.", text variable: m_instance.cfg.nSetpointTempTimeout, input disabled if: NOT m_instance.stat.bEngMode
            OnMouseClick: write the text variable via Default
    GroupBox (304,722 271x111), "Last forced switch to MANUAL"
        Label (10,30 61x21), "Time:"
        Label (10,50 61x21), "Cause"
        Rectangle (70,30 181x20), "%s", text variable: m_instance.stat.sLastForcedManualTime
        Rectangle (70,50 181x20), "%s", text variable: m_instance.stat.sLastForcedManualCause
        Button (70,80 181x21), "Clear diagnostics", input disabled if: NOT m_instance.stat.bEngMode
            OnMouseClick: execute { m_instance.ctrl.bClearForcedManualDiag := TRUE; }
    Ellipse (760,296 6x6)
END_VISUALIZATION

// HMI/VISUs/Templates/TEMPLATE_METIS_CTRL_TEMPERATURE_SIMPLIFIED
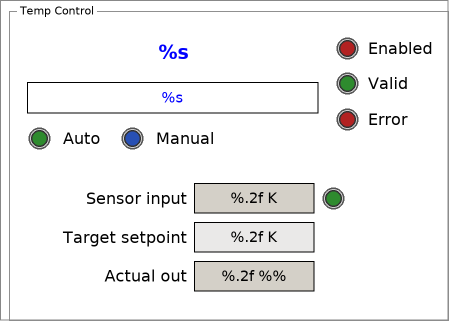
VISUALIZATION TEMPLATE_METIS_CTRL_TEMPERATURE_SIMPLIFIED  // 449x321
VAR_IN_OUT
	m_instance  : FB_METIS_CTRL_TEMPERATURE;
END_VAR
    GroupBox (9,3 440x318), "Temp Control"
    Group (20,33 419x258)
        Rectangle (0,2 308x35), "%s", text variable: m_instance.in_sName
        Group (38,189 256x31)
            Label (0,0 132x31), "Target setpoint"
            Rectangle (136,0 120x30), "%.2f K", tooltip "Target ramp setpoint", text variable: m_instance.stat.lrTargetSetpoint
        Group (315,71 80x31)
            Label (30,0 50x31), "Error"
            Lamp1 (0,3 25x25), variable: m_instance.stat.bError, style: Lamp-Lamp1-Red
        Rectangle (7,49 291x31), "%s", text variable: m_instance.stat.sStatus
        Group (72,228 222x30)
            Rectangle (102,0 120x30), "%.2f %%", tooltip "Set Velocity [UU/s]", text variable: m_instance.stat.lrControllerOut
            Label (0,0 98x30), "Actual out"
        Group (61,150 265x31)
            Label (0,0 109x31), "Sensor input"
            Rectangle (113,0 120x30), "%.2f K", tooltip "Actual input temperature", text variable: m_instance.stat.lrActInput
            Lamp1 (240,3 25x25), tooltip "Green if the input temperature is valid", variable: m_instance.stat.bActInputValid, style: Lamp-Lamp1-Green
        Group (315,35 81x31)
            Label (30,0 51x31), "Valid"
            Lamp1 (0,3 25x25), variable: m_instance.stat.bValid, style: Lamp-Lamp1-Green
        Group (7,90 81x31)
            Lamp1 (0,3 25x25), variable: m_instance.stat.bCtrlModeIsAuto, style: Lamp-Lamp1-Green
            Label (33,0 48x31), "Auto"
        Group (100,90 102x31)
            Lamp1 (0,3 25x25), variable: m_instance.stat.bCtrlModeIsManual, style: Lamp-Lamp1-Blue
            Label (33,0 69x31), "Manual"
        Group (315,0 104x31)
            Label (30,0 74x31), "Enabled"
            Lamp1 (0,3 25x25), variable: m_instance.cfg.bEnabled, style: Lamp-Lamp1-Red
END_VISUALIZATION

// HMI/VISUs/Templates/TEMPLATE_METIS_HEATER
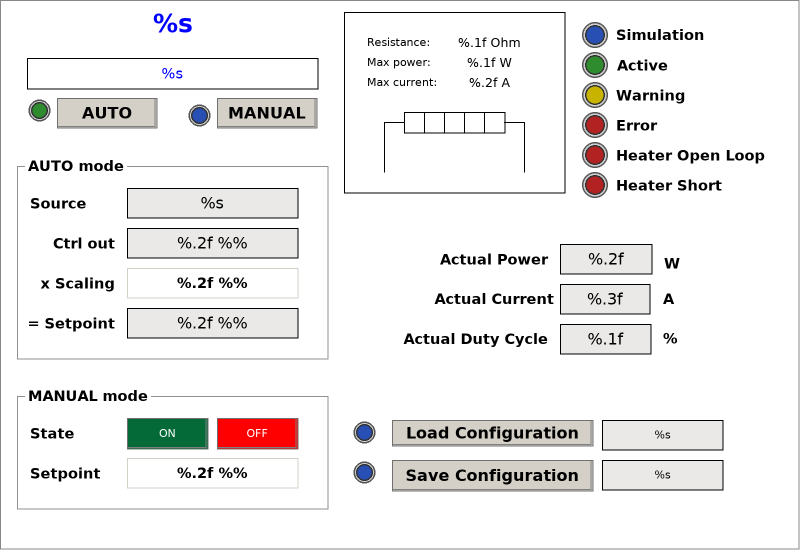
VISUALIZATION TEMPLATE_METIS_HEATER  // 800x550
VAR_IN_OUT
	m_instance: FB_METIS_HEATER;
END_VAR
    Rectangle (8,8 330x30), "%s", text variable: m_Instance.in_sName
    Group (580,20 184x180)
        Group (0,30 184x30)
            Lamp1 (0,0 30x30), tooltip "If ON, Heater is active", variable: m_Instance.stat.bActive, style: Lamp-Lamp1-Green
            Label (34,4 150x23), "Active"
        Group (0,60 183x30)
            Lamp1 (0,0 30x30), tooltip "If ON, reading is in Warning", variable: m_Instance.stat.bWarning, style: Lamp-Lamp1-Yellow
            Label (33,4 150x23), "Warning"
        Group (0,90 183x30)
            Lamp1 (0,0 30x30), tooltip "If ON, reading is in error.", variable: m_Instance.stat.bError, style: Lamp-Lamp1-Red
            Label (33,4 150x23), "Error"
        Group (0,120 183x30)
            Lamp1 (0,0 30x30), tooltip "If ON, Heater circuit is open", variable: m_Instance.stat.bHeaterOpenLoop, style: Lamp-Lamp1-Red
            Label (33,4 150x23), "Heater Open Loop"
        Group (0,150 183x30)
            Lamp1 (0,0 30x30), tooltip "If ON, Heater is in short circuit", variable: m_Instance.stat.bHeaterShort, style: Lamp-Lamp1-Red
            Label (33,4 150x23), "Heater Short"
        Group (0,0 143x30)
            Lamp1 (0,0 30x30), tooltip "If ON, Heater is simulated.", variable: m_instance.stat.bSimulated, style: Lamp-Lamp1-Blue
            Rectangle (33,0 110x30), "Simulation"
    Group (400,244 292x110)
        Rectangle (160,80 91x30), "%.1f", tooltip "Value used by the system [C]", text variable: m_instance.stat.lrActDutyCycle, invisible if: NOT m_instance.stat.bActDutyCycleAvailable
        Rectangle (0,80 151x30), "Actual Duty Cycle", invisible if: NOT m_instance.stat.bActDutyCycleAvailable
        Rectangle (160,0 92x30), "%.2f", tooltip "Value used by the system [K]", text variable: m_instance.stat.lrActHeaterPower
        Rectangle (160,40 90x30), "%.3f", tooltip "Value used by the system [C]", text variable: m_instance.stat.lrActCurrent
        Rectangle (261,5 29x29), "W"
        Rectangle (260,40 32x30), "A"
        Rectangle (40,0 111x31), "Actual Power"
        Rectangle (30,40 127x30), "Actual Current"
        Rectangle (260,79 29x31), "%", invisible if: NOT m_instance.stat.bActDutyCycleAvailable
    Group (344,12 221x181)
        Rectangle (0,0 221x181)
        Rectangle (60,100 101x21)
        Line (40,110) (60,110)
        Line (40,110) (40,160)
        Line (180,110) (180,160)
        Line (160,110) (180,110)
        Line (80,100) (80,120)
        Line (100,100) (100,120)
        Line (120,100) (120,120)
        Line (140,100) (140,120)
        Label (20,20 81x21), "Resistance:"
        Rectangle (90,20 111x21), "%.1f Ohm", tooltip "Value used by the system [K]", text variable: m_instance.in_lrHeaterResistance
        Label (20,40 81x21), "Max power:"
        Rectangle (90,40 111x21), "%.1f W", tooltip "Value used by the system [K]", text variable: m_instance.in_lrHeaterMaxPower
        Label (20,60 81x21), "Max current:"
        Rectangle (90,60 111x21), "%.2f A", tooltip "Value used by the system [K]", text variable: m_instance.stat.lrMaxCurrent
    GroupBox (17,388 311x121), "MANUAL mode"
        Rectangle (10,30 131x31), "State"
        Rectangle (10,70 101x31), "Setpoint"
        Button (110,30 81x31), "ON", input disabled if: NOT m_instance.stat.bManual
            OnMouseClick: execute { m_instance.ctrl.bManualEnable := TRUE; }
        Button (200,30 81x31), "OFF", input disabled if: NOT m_instance.stat.bManual
            OnMouseClick: execute { m_instance.ctrl.bManualEnable := FALSE; }
        Textfield (110,70 171x30), "%.2f %%", text variable: m_instance.ctrl.lrManualSetpoint, input disabled if: NOT m_instance.stat.bManual
            OnMouseClick: write the text variable via Default
    Lamp1 (187,103 25x25), variable: m_instance.stat.bManual, style: Lamp-Lamp1-Blue
    Lamp1 (27,98 25x25), variable: m_instance.stat.bAuto, style: Lamp-Lamp1-Green
    Button (57,98 100x30), "AUTO", tooltip "Switch to AUTO Mode", input disabled if: NOT m_instance.stat.bAcceptCtrlMode_Auto
        OnMouseClick: execute { m_instance.ctrl.eCtrlMode := E_METIS_CTRL_MODE.AUTO; }
    Button (217,98 100x30), "MANUAL", tooltip "Switch to MANUAL Mode", input disabled if: NOT m_instance.stat.bAcceptCtrlMode_Manual
        OnMouseClick: execute { m_instance.ctrl.eCtrlMode := E_METIS_CTRL_MODE.MANUAL; }
    Rectangle (27,58 291x31), "%s", text variable: m_Instance.stat.sHeaterState
    Lamp1 (352,420 25x25), tooltip "Command coming from the Control System", variable: m_instance.ctrl.bReadConfig, style: Lamp-Lamp1-Blue
    Button (392,460 201x31), "Save Configuration"
        OnMouseClick: execute { m_instance.ctrl.bWriteConfig := TRUE; }
    Button (392,420 201x26), "Load Configuration"
        OnMouseClick: execute { m_instance.ctrl.bReadConfig := TRUE; }
    Lamp1 (352,460 25x25), tooltip "Command coming from the Control System", variable: m_instance.ctrl.bWriteConfig, style: Lamp-Lamp1-Blue
    Rectangle (602,420 121x30), "%s", text variable: m_Instance.fbConfig.sReadError, colour toggle: m_Instance.fbConfig.bReadError
    Rectangle (602,460 121x30), "%s", text variable: m_Instance.fbConfig.sWriteError, colour toggle: m_Instance.fbConfig.bWriteError
    GroupBox (17,158 311x201), "AUTO mode"
        Rectangle (110,30 171x30), "%s", tooltip "Value used by the system [C]", text variable: m_instance.stat.sAutoSetpointSource
        Rectangle (10,30 91x31), "Source"
        Rectangle (10,150 91x31), "= Setpoint", tooltip "Setpoint after the scaling was applied"
        Rectangle (110,150 171x30), "%.2f %%", tooltip "Value used by the system [C]", text variable: m_instance.stat.lrAutoSetpointValue
        Textfield (110,110 171x30), "%.2f %%", text variable: m_instance.cfg.lrAutoScalePercent
            OnMouseClick: write the text variable via Default
        Rectangle (10,110 91x31), "x Scaling", tooltip "Setpoint = controller output x scaling"
        Rectangle (110,70 171x30), "%.2f %%", tooltip "Value used by the system [C]", text variable: m_instance.stat.lrAutoCtrlOut
        Rectangle (10,70 91x31), "Ctrl out", tooltip "Setpoint = controller output x scaling"
END_VISUALIZATION

// HMI/VISUs/Templates/TEMPLATE_METIS_HEATER_SIMPLIFIED
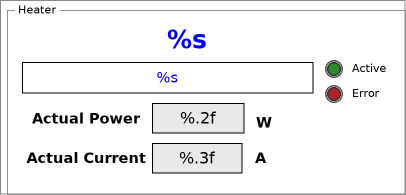
VISUALIZATION TEMPLATE_METIS_HEATER_SIMPLIFIED  // 406x195
VAR_IN_OUT
	m_instance: FB_METIS_HEATER;
END_VAR
    GroupBox (7,2 399x193), "Heater"
    Group (22,24 369x149)
        Lamp1 (302,35 20x20), tooltip "If ON, Heater is active", variable: m_Instance.stat.bActive, style: Lamp-Lamp1-Green
        Rectangle (0,0 330x30), "%s", text variable: m_Instance.in_sName
        Lamp1 (302,60 20x20), tooltip "If ON, reading is in error.", variable: m_Instance.stat.bError, style: Lamp-Lamp1-Red
        Label (327,33 42x23), "Active"
        Label (327,58 36x23), "Error"
        Group (0,79 262x70)
            Rectangle (130,0 92x30), "%.2f", tooltip "Value used by the system [K]", text variable: m_instance.stat.lrActHeaterPower
            Rectangle (130,40 90x30), "%.3f", tooltip "Value used by the system [C]", text variable: m_instance.stat.lrActCurrent
            Rectangle (231,5 29x29), "W"
            Rectangle (230,40 32x30), "A"
            Rectangle (10,0 111x31), "Actual Power"
            Rectangle (0,40 127x30), "Actual Current"
        Rectangle (0,38 291x31), "%s", text variable: m_Instance.stat.sHeaterState
END_VISUALIZATION

// HMI/VISUs/Templates/TEMPLATE_PRESSURE_READING
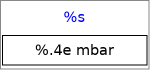
VISUALIZATION TEMPLATE_PRESSURE_READING  // 150x70
VAR_IN_OUT
	m_instance: FB_CRYO_SENSOR_PRESSURE;
END_VAR
    Rectangle (2,35 145x30), "%.4e mbar", tooltip "Pressure in mbar", text variable: m_instance.stat.lrPressure, colour toggle: NOT m_instance.stat.bValid
    Rectangle (2,2 145x30), "%s", text variable: m_instance.in_sName
END_VISUALIZATION

// HMI/VISUs/Templates/TEMPLATE_RESET_VALVES
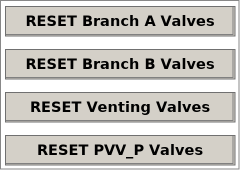
VISUALIZATION TEMPLATE_RESET_VALVES  // 240x170
VAR_IN_OUT
	m_instance_evac_branch_A:	FB_CRYO_EVAC_BRANCH_A;
	m_instance_evac_branch_B:	FB_CRYO_EVAC_BRANCH_B;
	m_instance_venting:			FB_METIS_CRYO_VENTING;
	m_instance_cool_down:		FB_METIS_CRYO_COOL_DOWN;
END_VAR
    Button (5,6 230x30), "RESET Branch A Valves"
        OnMouseClick: execute { m_instance_evac_branch_A.bReset_Valves := TRUE; }
    Button (5,49 230x30), "RESET Branch B Valves"
        OnMouseClick: execute { m_instance_evac_branch_B.bReset_Valves := TRUE; }
    Button (5,92 230x30), "RESET Venting Valves"
        OnMouseClick: execute { m_instance_venting.bReset_Valves := TRUE; }
    Button (5,135 230x30), "RESET PVV_P Valves"
        OnMouseClick: execute { m_instance_cool_down.bReset_Valves := TRUE; }
END_VISUALIZATION

// HMI/VISUs/Templates/TEMPLATE_TEMP_SENSOR_VALUE_ONLY
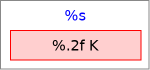
VISUALIZATION TEMPLATE_TEMP_SENSOR_VALUE_ONLY  // 150x70
VAR_IN_OUT
	m_instance:	FB_METIS_TEMPERATURE;
	
END_VAR
    Rectangle (10,30 131x30)
    Rectangle (10,30 131x30), invisible if: NOT m_instance.stat.bWarning
    Rectangle (10,30 131x30), invisible if: NOT m_instance.stat.bError
    Rectangle (10,30 131x31), "%.2f K", tooltip "%s", text variable: m_instance.stat.lrTempK
        p4168582468: m_instance.stat.sErrorText
    Rectangle (0,0 151x31), "%s", text variable: m_instance.stat.sName
END_VISUALIZATION

// HMI/VISUs/Templates/TEMPLATE_TEMPERATURE_VOTE
